C01825=1176.377,-89.170,-41.467,179.123,5.741,149.280
C01826=1176.382,-89.420,-41.456,179.120,5.741,149.280
C01827=1176.387,-89.669,-41.446,179.119,5.741,149.281
C01828=1176.393,-89.919,-41.437,179.116,5.740,149.282
C01829=1176.399,-90.169,-41.427,179.114,5.739,149.282
C01830=1176.403,-90.419,-41.417,179.112,5.740,149.283
C01831=1176.409,-90.668,-41.406,179.110,5.739,149.283
C01832=1176.414,-90.918,-41.396,179.108,5.739,149.284
C01833=1176.419,-91.168,-41.387,179.105,5.739,149.285
C01834=1176.424,-91.418,-41.377,179.103,5.738,149.285
C01835=1176.430,-91.668,-41.367,179.101,5.739,149.286
C01836=1176.435,-91.917,-41.357,179.098,5.738,149.286
C01837=1176.441,-92.167,-41.347,179.096,5.738,149.287
C01838=1176.446,-92.417,-41.337,179.094,5.738,149.288
C01839=1176.451,-92.666,-41.327,179.092,5.737,149.288
C01840=1176.456,-92.916,-41.317,179.090,5.737,149.289
C01841=1176.462,-93.166,-41.308,179.087,5.737,149.290
C01842=1176.467,-93.415,-41.298,179.086,5.737,149.290
C01843=1176.472,-93.666,-41.287,179.083,5.736,149.291
C01844=1176.478,-93.915,-41.277,179.081,5.736,149.291
C01845=1176.483,-94.165,-41.268,179.079,5.736,149.292
C01846=1176.488,-94.415,-41.258,179.077,5.735,149.292
C01847=1176.493,-94.664,-41.248,179.074,5.736,149.293
C01848=1176.499,-94.915,-41.239,179.072,5.735,149.294
C01849=1176.504,-95.164,-41.228,179.070,5.734,149.294
C01850=1176.509,-95.413,-41.219,179.068,5.734,149.295
C01851=1176.515,-95.664,-41.209,179.065,5.734,149.296
C01852=1176.520,-95.913,-41.200,179.064,5.734,149.296
C01853=1176.525,-96.162,-41.189,179.061,5.734,149.297
C01854=1176.531,-96.413,-41.180,179.059,5.734,149.297
C01855=1176.536,-96.663,-41.170,179.057,5.733,149.298
C01856=1176.541,-96.912,-41.160,179.055,5.733,149.298
C01857=1176.546,-97.162,-41.151,179.053,5.733,149.299
C01858=1176.552,-97.411,-41.141,179.050,5.732,149.300
C01859=1176.557,-97.661,-41.132,179.048,5.733,149.300
C01860=1176.562,-97.912,-41.121,179.046,5.732,149.301
C01861=1176.568,-98.161,-41.111,179.044,5.732,149.302
C01862=1176.573,-98.411,-41.102,179.042,5.731,149.302
C01863=1176.578,-98.660,-41.092,179.039,5.731,149.303
C01864=1176.584,-98.910,-41.083,179.038,5.731,149.303
C01865=1176.589,-99.160,-41.073,179.035,5.731,149.304
C01866=1176.594,-99.410,-41.064,179.033,5.731,149.304
C01867=1176.600,-99.659,-41.054,179.031,5.730,149.305
C01868=1176.604,-99.909,-41.044,179.029,5.730,149.306
C01869=1176.610,-100.159,-41.034,179.026,5.730,149.306
C01870=1176.615,-100.409,-41.025,179.024,5.729,149.307
C01871=1176.621,-100.659,-41.015,179.022,5.729,149.308
C01872=1176.626,-100.908,-41.005,179.020,5.729,149.308
C01873=1176.632,-101.158,-40.996,179.018,5.729,149.309
C01874=1176.636,-101.407,-40.986,179.016,5.728,149.309
C01875=1176.643,-101.680,-40.976,179.013,5.728,149.310
C01876=1176.648,-101.952,-40.965,179.011,5.728,149.311
C01877=1176.654,-102.223,-40.955,179.009,5.728,149.311
C01878=1176.660,-102.495,-40.945,179.006,5.727,149.312
C01879=1176.665,-102.745,-40.935,179.004,5.728,149.313
C01880=1176.670,-102.995,-40.926,179.002,5.727,149.313
C01881=1176.676,-103.244,-40.916,179.000,5.727,149.314
C01882=1176.681,-103.494,-40.907,178.997,5.726,149.314
C01883=1176.686,-103.743,-40.897,178.996,5.726,149.315
C01884=1176.691,-103.994,-40.888,178.993,5.726,149.315
C01885=1176.696,-104.243,-40.878,178.992,5.726,149.316
C01886=1176.702,-104.493,-40.868,178.989,5.726,149.317
C01887=1176.707,-104.743,-40.860,178.987,5.725,149.317
C01888=1176.713,-104.992,-40.849,178.985,5.725,149.318
C01889=1176.718,-105.242,-40.840,178.982,5.725,149.318
C01890=1176.723,-105.491,-40.831,178.980,5.725,149.319
C01891=1176.729,-105.742,-40.821,178.978,5.724,149.319
C01892=1176.734,-105.991,-40.812,178.976,5.725,149.320
C01893=1176.740,-106.241,-40.802,178.974,5.724,149.321
C01894=1176.745,-106.491,-40.793,178.972,5.724,149.321
C01895=1176.749,-106.741,-40.783,178.970,5.723,149.322
C01896=1176.755,-106.991,-40.774,178.967,5.723,149.323
C01897=1176.760,-107.241,-40.765,178.965,5.723,149.323
C01898=1176.765,-107.490,-40.755,178.963,5.723,149.324
C01899=1176.771,-107.740,-40.746,178.961,5.723,149.324
C01900=1176.776,-107.990,-40.737,178.959,5.722,149.325
C01901=1176.781,-108.239,-40.727,178.957,5.722,149.325
C01902=1176.787,-108.489,-40.718,178.955,5.722,149.326
C01903=1176.792,-108.739,-40.709,178.952,5.722,149.327
C01904=1176.797,-108.989,-40.699,178.950,5.721,149.327
C01905=1176.803,-109.239,-40.690,178.948,5.722,149.328
C01906=1176.808,-109.489,-40.681,178.946,5.721,149.328
C01907=1176.813,-109.738,-40.672,178.944,5.721,149.329
C01908=1176.819,-109.988,-40.662,178.942,5.721,149.330
C01909=1176.824,-110.238,-40.653,178.940,5.721,149.330
C01910=1176.829,-110.488,-40.644,178.937,5.720,149.331
C01911=1176.835,-110.737,-40.634,178.935,5.719,149.331
C01912=1176.840,-110.987,-40.625,178.933,5.720,149.332
C01913=1176.845,-111.237,-40.616,178.931,5.719,149.332
C01914=1176.851,-111.487,-40.607,178.929,5.719,149.333
C01915=1176.856,-111.737,-40.598,178.927,5.719,149.334
C01916=1176.862,-111.985,-40.588,178.925,5.719,149.334
C01917=1176.867,-112.235,-40.579,178.922,5.718,149.335
C01918=1176.873,-112.485,-40.570,178.920,5.719,149.336
C01919=1176.878,-112.735,-40.561,178.918,5.718,149.336
C01920=1176.883,-112.985,-40.551,178.917,5.718,149.337
C01921=1176.889,-113.235,-40.542,178.914,5.718,149.337
C01922=1176.894,-113.485,-40.533,178.912,5.718,149.338
C01923=1176.899,-113.734,-40.524,178.910,5.717,149.338
C01924=1176.904,-113.984,-40.515,178.908,5.717,149.339
C01925=1176.910,-114.234,-40.506,178.905,5.717,149.340
C01926=1176.915,-114.484,-40.496,178.904,5.717,149.340
C01927=1176.920,-114.733,-40.487,178.901,5.716,149.341
C01928=1176.925,-114.983,-40.478,178.899,5.717,149.341
C01929=1176.931,-115.234,-40.469,178.897,5.716,149.342
C01930=1176.936,-115.483,-40.460,178.895,5.716,149.343
C01931=1176.941,-115.733,-40.451,178.893,5.715,149.343
C01932=1176.947,-115.982,-40.442,178.891,5.716,149.344
C01933=1176.952,-116.232,-40.433,178.889,5.715,149.344
C01934=1176.958,-116.482,-40.423,178.886,5.714,149.345
C01935=1176.963,-116.732,-40.415,178.884,5.715,149.345
C01936=1176.968,-116.981,-40.406,178.882,5.714,149.346
C01937=1176.973,-117.231,-40.397,178.880,5.714,149.347
C01938=1176.979,-117.481,-40.388,178.878,5.714,149.347
C01939=1176.984,-117.731,-40.379,178.876,5.714,149.348
C01940=1176.990,-117.981,-40.369,178.874,5.713,149.348
C01941=1176.995,-118.231,-40.361,178.872,5.713,149.349
C01942=1177.001,-118.480,-40.352,178.869,5.713,149.350
C01943=1177.006,-118.730,-40.343,178.868,5.713,149.350
C01944=1177.011,-118.979,-40.334,178.865,5.713,149.351
C01945=1177.016,-119.229,-40.325,178.863,5.713,149.351
C01946=1177.022,-119.479,-40.315,178.861,5.712,149.352
C01947=1177.027,-119.729,-40.306,178.859,5.712,149.352
C01948=1177.032,-119.979,-40.297,178.857,5.711,149.353
C01949=1177.037,-120.229,-40.288,178.855,5.712,149.354
C01950=1177.043,-120.478,-40.280,178.853,5.711,149.354
C01951=1177.048,-120.728,-40.271,178.851,5.711,149.355
C01952=1177.053,-120.978,-40.262,178.848,5.711,149.355
C01953=1177.058,-121.228,-40.253,178.847,5.711,149.356
C01954=1177.064,-121.477,-40.244,178.844,5.710,149.357
C01955=1177.070,-121.728,-40.235,178.843,5.710,149.357
C01956=1177.075,-121.977,-40.226,178.840,5.710,149.357
C01957=1177.080,-122.227,-40.217,178.838,5.710,149.358
C01958=1177.086,-122.476,-40.209,178.836,5.709,149.359
C01959=1177.091,-122.726,-40.200,178.834,5.710,149.359
C01960=1177.096,-122.977,-40.191,178.832,5.709,149.360
C01961=1177.101,-123.227,-40.183,178.830,5.709,149.360
C01962=1177.107,-123.476,-40.174,178.828,5.709,149.361
C01963=1177.112,-123.726,-40.165,178.826,5.709,149.362
C01964=1177.118,-123.975,-40.156,178.824,5.709,149.362
C01965=1177.123,-124.225,-40.147,178.822,5.708,149.363
C01966=1177.128,-124.475,-40.138,178.820,5.708,149.363
C01967=1177.133,-124.725,-40.130,178.817,5.708,149.364
C01968=1177.139,-124.974,-40.121,178.816,5.708,149.364
C01969=1177.144,-125.224,-40.112,178.814,5.707,149.365
C01970=1177.150,-125.474,-40.103,178.812,5.708,149.366
C01971=1177.155,-125.724,-40.094,178.809,5.707,149.366
C01972=1177.161,-125.974,-40.086,178.807,5.707,149.367
C01973=1177.166,-126.224,-40.077,178.805,5.706,149.367
C01974=1177.171,-126.473,-40.068,178.803,5.706,149.368
C01975=1177.177,-126.723,-40.059,178.801,5.706,149.369
C01976=1177.182,-126.973,-40.050,178.799,5.706,149.369
C01977=1177.188,-127.222,-40.042,178.797,5.705,149.370
C01978=1177.193,-127.473,-40.034,178.795,5.706,149.370
C01979=1176.771,-127.484,-40.074,178.791,5.709,149.372
C01980=1176.766,-127.234,-40.083,178.793,5.709,149.371
C01981=1176.761,-126.984,-40.091,178.795,5.709,149.371
C01982=1176.756,-126.734,-40.100,178.797,5.709,149.370
C01983=1176.750,-126.485,-40.108,178.800,5.710,149.370
C01984=1176.745,-126.235,-40.117,178.801,5.710,149.369
C01985=1176.739,-125.985,-40.126,178.803,5.710,149.369
C01986=1176.734,-125.735,-40.135,178.805,5.710,149.368
C01987=1176.729,-125.485,-40.144,178.808,5.711,149.368
C01988=1176.723,-125.236,-40.152,178.810,5.710,149.367
C01989=1176.718,-124.986,-40.160,178.812,5.711,149.366
C01990=1176.713,-124.736,-40.169,178.814,5.711,149.366
C01991=1176.707,-124.486,-40.179,178.816,5.711,149.365
C01992=1176.702,-124.236,-40.188,178.818,5.711,149.365
C01993=1176.696,-123.987,-40.196,178.820,5.712,149.364
C01994=1176.691,-123.737,-40.205,178.822,5.712,149.363
C01995=1176.685,-123.487,-40.214,178.824,5.713,149.363
C01996=1176.680,-123.237,-40.223,178.826,5.712,149.362
C01997=1176.675,-122.987,-40.232,178.829,5.713,149.362
C01998=1176.670,-122.737,-40.241,178.830,5.713,149.361
C01999=1176.664,-122.488,-40.249,178.833,5.713,149.361
C02000=1176.659,-122.238,-40.257,178.834,5.713,149.360
C02001=1176.654,-121.988,-40.266,178.837,5.714,149.360
C02002=1176.648,-121.738,-40.275,178.839,5.714,149.359
C02003=1176.643,-121.488,-40.284,178.841,5.714,149.358
C02004=1176.638,-121.238,-40.293,178.843,5.714,149.358
C02005=1176.632,-120.989,-40.302,178.845,5.715,149.357
C02006=1176.626,-120.739,-40.311,178.847,5.715,149.357
C02007=1176.621,-120.489,-40.320,178.849,5.715,149.356
C02008=1176.616,-120.239,-40.329,178.851,5.715,149.355
C02009=1176.611,-119.990,-40.338,178.854,5.715,149.355
C02010=1176.606,-119.740,-40.347,178.855,5.715,149.354
C02011=1176.601,-119.490,-40.356,178.858,5.716,149.354
C02012=1176.595,-119.241,-40.364,178.860,5.716,149.353
C02013=1176.589,-118.991,-40.374,178.862,5.717,149.353
C02014=1176.584,-118.741,-40.383,178.864,5.716,149.352
C02015=1176.579,-118.491,-40.392,178.866,5.717,149.351
C02016=1176.574,-118.242,-40.401,178.868,5.717,149.351
C02017=1176.569,-117.992,-40.410,178.870,5.717,149.350
C02018=1176.563,-117.742,-40.419,178.872,5.717,149.350
C02019=1176.558,-117.492,-40.428,178.875,5.718,149.349
C02020=1176.552,-117.242,-40.437,178.876,5.718,149.348
C02021=1176.547,-116.993,-40.446,178.879,5.718,149.348
C02022=1176.541,-116.743,-40.455,178.880,5.718,149.347
C02023=1176.536,-116.493,-40.464,178.883,5.719,149.347
C02024=1176.531,-116.243,-40.472,178.885,5.718,149.346
C02025=1176.525,-115.993,-40.482,178.887,5.719,149.346
C02026=1176.520,-115.744,-40.492,178.889,5.719,149.345
C02027=1176.515,-115.494,-40.500,178.891,5.719,149.344
C02028=1176.510,-115.244,-40.509,178.893,5.719,149.344
C02029=1176.505,-114.994,-40.518,178.896,5.720,149.343
C02030=1176.499,-114.744,-40.528,178.897,5.720,149.343
C02031=1176.494,-114.494,-40.537,178.900,5.720,149.342
C02032=1176.488,-114.245,-40.545,178.901,5.720,149.342
C02033=1176.483,-113.996,-40.555,178.904,5.720,149.341
C02034=1176.477,-113.746,-40.564,178.906,5.720,149.340
C02035=1176.472,-113.496,-40.573,178.908,5.721,149.340
C02036=1176.467,-113.246,-40.582,178.910,5.721,149.339
C02037=1176.462,-112.996,-40.591,178.912,5.722,149.339
C02038=1176.456,-112.747,-40.601,178.914,5.721,149.338
C02039=1176.451,-112.497,-40.610,178.916,5.722,149.337
C02040=1176.446,-112.247,-40.619,178.919,5.722,149.337
C02041=1176.440,-111.997,-40.628,178.921,5.722,149.336
C02042=1176.435,-111.747,-40.637,178.923,5.723,149.336
C02043=1176.430,-111.498,-40.647,178.925,5.723,149.335
C02044=1176.425,-111.248,-40.656,178.927,5.723,149.335
C02045=1176.419,-110.998,-40.665,178.929,5.723,149.334
C02046=1176.414,-110.748,-40.674,178.931,5.724,149.333
C02047=1176.409,-110.499,-40.684,178.934,5.723,149.333
C02048=1176.403,-110.248,-40.693,178.936,5.724,149.332
C02049=1176.398,-109.999,-40.702,178.938,5.724,149.331
C02050=1176.392,-109.749,-40.711,178.940,5.725,149.331
C02051=1176.387,-109.499,-40.721,178.942,5.724,149.330
C02052=1176.382,-109.249,-40.730,178.944,5.725,149.330
C02053=1176.377,-108.999,-40.739,178.946,5.725,149.329
C02054=1176.371,-108.750,-40.749,178.949,5.725,149.329
C02055=1176.366,-108.500,-40.758,178.951,5.726,149.328
C02056=1176.361,-108.250,-40.767,178.953,5.726,149.327
C02057=1176.355,-108.001,-40.777,178.955,5.726,149.327
C02058=1176.350,-107.751,-40.786,178.957,5.726,149.326
C02059=1176.345,-107.501,-40.795,178.959,5.727,149.326
C02060=1176.339,-107.251,-40.805,178.961,5.726,149.325
C02061=1176.334,-107.002,-40.814,178.964,5.727,149.324
C02062=1176.329,-106.752,-40.823,178.965,5.727,149.324
C02063=1176.323,-106.502,-40.833,178.968,5.727,149.323
C02064=1176.318,-106.252,-40.842,178.969,5.727,149.323
C02065=1176.313,-106.002,-40.851,178.972,5.728,149.322
C02066=1176.307,-105.753,-40.861,178.974,5.728,149.322
C02067=1176.302,-105.503,-40.870,178.976,5.728,149.321
C02068=1176.296,-105.254,-40.880,178.979,5.729,149.320
C02069=1176.291,-105.004,-40.889,178.981,5.729,149.320
C02070=1176.286,-104.754,-40.898,178.983,5.729,149.319
C02071=1176.281,-104.504,-40.909,178.985,5.729,149.318
C02072=1176.275,-104.254,-40.917,178.987,5.730,149.318
C02073=1176.270,-104.005,-40.928,178.989,5.729,149.317
C02074=1176.265,-103.754,-40.937,178.991,5.730,149.317
C02075=1176.260,-103.505,-40.947,178.993,5.730,149.316
C02076=1176.254,-103.255,-40.956,178.996,5.730,149.316
C02077=1176.249,-103.005,-40.965,178.998,5.731,149.315
C02078=1176.244,-102.756,-40.975,179.000,5.731,149.314
C02079=1176.239,-102.506,-40.984,179.002,5.732,149.314
C02080=1176.232,-102.233,-40.995,179.004,5.731,149.313
C02081=1176.226,-101.963,-41.005,179.007,5.732,149.312
C02082=1176.221,-101.691,-41.016,179.010,5.732,149.312
C02083=1176.216,-101.419,-41.026,179.011,5.732,149.311
C02084=1176.210,-101.169,-41.035,179.014,5.732,149.311
C02085=1176.205,-100.920,-41.045,179.016,5.733,149.310
C02086=1176.199,-100.669,-41.054,179.018,5.733,149.309
C02087=1176.194,-100.420,-41.064,179.020,5.733,149.309
C02088=1176.189,-100.170,-41.075,179.022,5.733,149.308
C02089=1176.184,-99.920,-41.084,179.025,5.734,149.308
C02090=1176.178,-99.671,-41.094,179.027,5.733,149.307
C02091=1176.173,-99.421,-41.103,179.029,5.734,149.306
C02092=1176.167,-99.171,-41.113,179.032,5.735,149.306
C02093=1176.162,-98.921,-41.122,179.033,5.735,149.305
C02094=1176.157,-98.672,-41.132,179.036,5.735,149.305
C02095=1176.152,-98.422,-41.141,179.037,5.735,149.304
C02096=1176.147,-98.172,-41.151,179.040,5.735,149.303
C02097=1176.142,-97.922,-41.161,179.042,5.735,149.303
C02098=1176.136,-97.672,-41.171,179.044,5.736,149.302
C02099=1176.130,-97.423,-41.181,179.047,5.737,149.302
C02100=1176.125,-97.173,-41.190,179.049,5.736,149.301
C02101=1176.119,-96.923,-41.200,179.051,5.737,149.300
C02102=1176.115,-96.674,-41.209,179.053,5.736,149.300
C02103=1176.109,-96.423,-41.219,179.055,5.737,149.299
C02104=1176.104,-96.174,-41.229,179.057,5.737,149.299
C02105=1176.099,-95.924,-41.239,179.059,5.738,149.298
C02106=1176.093,-95.674,-41.249,179.062,5.738,149.297
C02107=1176.088,-95.425,-41.258,179.064,5.738,149.297
C02108=1176.082,-95.176,-41.268,179.066,5.738,149.296
C02109=1176.078,-94.925,-41.278,179.068,5.738,149.296
C02110=1176.072,-94.675,-41.288,179.071,5.739,149.295
C02111=1176.067,-94.426,-41.298,179.073,5.740,149.295
C02112=1176.061,-94.176,-41.307,179.075,5.739,149.294
C02113=1176.056,-93.927,-41.317,179.077,5.740,149.293
C02114=1176.051,-93.676,-41.328,179.079,5.740,149.293
C02115=1176.046,-93.426,-41.337,179.081,5.740,149.292
C02116=1176.040,-93.177,-41.347,179.083,5.740,149.291
C02117=1176.035,-92.928,-41.357,179.086,5.741,149.291
C02118=1176.030,-92.678,-41.367,179.088,5.741,149.290
C02119=1176.024,-92.427,-41.377,179.090,5.741,149.290
C02120=1176.020,-92.178,-41.386,179.093,5.741,149.289
C02121=1176.014,-91.928,-41.396,179.094,5.741,149.289
C02122=1176.008,-91.679,-41.407,179.097,5.742,149.288
C02123=1176.004,-91.428,-41.416,179.099,5.743,149.287
C02124=1175.998,-91.179,-41.426,179.101,5.742,149.287
C02125=1175.993,-90.929,-41.436,179.103,5.743,149.286
C02126=1175.988,-90.680,-41.446,179.105,5.743,149.285
C02127=1175.982,-90.429,-41.456,179.108,5.743,149.285
C02128=1175.977,-90.180,-41.466,179.110,5.744,149.284
C02129=1175.972,-89.930,-41.476,179.112,5.743,149.284
C02130=1175.966,-89.681,-41.486,179.114,5.744,149.283
C02131=1175.961,-89.431,-41.496,179.117,5.744,149.282
C02132=1175.955,-89.180,-41.506,179.119,5.745,149.282
C02133=1175.951,-88.931,-41.515,179.121,5.745,149.281
C02134=1175.945,-88.682,-41.526,179.123,5.745,149.281
C02135=1175.940,-88.431,-41.536,179.126,5.745,149.280
C02136=1175.935,-88.182,-41.546,179.127,5.745,149.279
C02137=1175.930,-87.933,-41.556,179.130,5.746,149.279
C02138=1175.924,-87.683,-41.566,179.132,5.747,149.278
C02139=1175.919,-87.432,-41.576,179.134,5.746,149.278
C02140=1175.914,-87.183,-41.586,179.136,5.747,149.277
C02141=1175.908,-86.933,-41.596,179.139,5.747,149.276
C02142=1175.903,-86.683,-41.607,179.141,5.747,149.276
C02143=1175.898,-86.434,-41.617,179.143,5.748,149.275
C02144=1175.893,-86.184,-41.626,179.145,5.747,149.274
C02145=1175.888,-85.934,-41.637,179.148,5.748,149.274
C02146=1175.882,-85.685,-41.647,179.150,5.748,149.273
C02147=1175.876,-85.435,-41.657,179.152,5.748,149.273
C02148=1175.871,-85.186,-41.668,179.155,5.749,149.272
C02149=1175.867,-84.936,-41.678,179.157,5.750,149.272
C02150=1175.861,-84.686,-41.688,179.159,5.749,149.271
C02151=1175.855,-84.437,-41.698,179.161,5.750,149.270
C02152=1175.850,-84.186,-41.708,179.163,5.750,149.270
C02153=1175.845,-83.936,-41.718,179.165,5.750,149.269
C02154=1175.840,-83.687,-41.728,179.168,5.751,149.269
C02155=1175.835,-83.437,-41.738,179.170,5.750,149.268
C02156=1175.829,-83.187,-41.748,179.172,5.751,149.267
C02157=1175.823,-82.938,-41.759,179.175,5.752,149.267
C02158=1175.818,-82.687,-41.769,179.177,5.752,149.266
C02159=1175.813,-82.438,-41.779,179.179,5.752,149.265
C02160=1175.809,-82.188,-41.789,179.181,5.752,149.265
C02161=1175.803,-81.938,-41.800,179.183,5.752,149.264
C02162=1175.798,-81.689,-41.811,179.186,5.753,149.264
C02163=1175.793,-81.439,-41.821,179.188,5.753,149.263
C02164=1175.787,-81.190,-41.831,179.190,5.754,149.263
C02165=1175.782,-80.940,-41.842,179.193,5.754,149.262
C02166=1175.777,-80.690,-41.852,179.195,5.754,149.261
C02167=1175.771,-80.440,-41.862,179.197,5.754,149.261
C02168=1175.766,-80.191,-41.872,179.200,5.755,149.260
C02169=1175.761,-79.941,-41.883,179.201,5.755,149.259
C02170=1175.755,-79.691,-41.893,179.204,5.755,149.259
C02171=1175.750,-79.441,-41.903,179.205,5.755,149.258
C02172=1175.745,-79.191,-41.914,179.208,5.756,149.258
C02173=1175.739,-78.942,-41.924,179.211,5.756,149.257
C02174=1175.734,-78.692,-41.934,179.212,5.756,149.256
C02175=1175.729,-78.443,-41.945,179.215,5.756,149.256
C02176=1175.724,-78.193,-41.956,179.217,5.757,149.255
C02177=1175.718,-77.943,-41.966,179.219,5.757,149.254
C02178=1175.713,-77.693,-41.976,179.221,5.758,149.254
C02179=1175.708,-77.443,-41.987,179.224,5.758,149.253
C02180=1175.702,-77.194,-41.997,179.226,5.758,149.253
C02181=1175.697,-76.943,-42.008,179.228,5.758,149.252
C02182=1175.692,-76.694,-42.018,179.231,5.759,149.251
C02183=1175.687,-76.444,-42.029,179.233,5.759,149.251
C02184=1175.681,-76.174,-42.040,179.235,5.759,149.250
C02185=1175.675,-75.902,-42.051,179.238,5.760,149.249
C02186=1175.670,-75.632,-42.062,179.241,5.760,149.249
C02187=1175.664,-75.360,-42.074,179.242,5.760,149.248
C02188=1175.659,-75.110,-42.085,179.245,5.760,149.248
C02189=1175.654,-74.861,-42.095,179.247,5.761,149.247
C02190=1175.649,-74.611,-42.106,179.249,5.761,149.246
C02191=1175.643,-74.361,-42.116,179.252,5.761,149.246
C02192=1175.637,-74.112,-42.126,179.254,5.762,149.245
C02193=1175.632,-73.862,-42.137,179.256,5.762,149.245
C02194=1175.627,-73.613,-42.148,179.258,5.762,149.244
C02195=1175.622,-73.363,-42.159,179.261,5.763,149.243
C02196=1175.616,-73.113,-42.169,179.263,5.762,149.243
C02197=1175.612,-72.863,-42.180,179.265,5.763,149.242
C02198=1175.606,-72.614,-42.190,179.268,5.764,149.241
C02199=1175.601,-72.364,-42.201,179.270,5.764,149.241
C02200=1175.596,-72.114,-42.211,179.272,5.764,149.240
C02201=1175.591,-71.864,-42.222,179.274,5.765,149.240
C02202=1175.585,-71.615,-42.233,179.276,5.764,149.239
C02203=1175.580,-71.364,-42.244,179.279,5.765,149.238
C02204=1175.574,-71.115,-42.255,179.281,5.766,149.238
C02205=1175.569,-70.865,-42.265,179.283,5.765,149.237
C02206=1175.564,-70.616,-42.275,179.286,5.766,149.237
C02207=1175.559,-70.366,-42.287,179.288,5.766,149.236
C02208=1175.553,-70.116,-42.297,179.291,5.767,149.235
C02209=1175.548,-69.866,-42.307,179.293,5.767,149.235
C02210=1175.543,-69.617,-42.318,179.295,5.767,149.234
C02211=1175.538,-69.367,-42.329,179.297,5.768,149.234
C02212=1175.533,-69.118,-42.340,179.299,5.768,149.233
C02213=1175.527,-68.868,-42.351,179.302,5.768,149.232
C02214=1175.521,-68.618,-42.361,179.304,5.769,149.232
C02215=1175.517,-68.368,-42.373,179.306,5.768,149.231
C02216=1175.511,-68.119,-42.383,179.309,5.769,149.231
C02217=1175.506,-67.869,-42.394,179.311,5.770,149.230
C02218=1175.501,-67.619,-42.405,179.313,5.770,149.229
C02219=1175.496,-67.369,-42.415,179.316,5.770,149.229
C02220=1175.490,-67.119,-42.427,179.318,5.770,149.228
C02221=1175.485,-66.870,-42.437,179.320,5.770,149.227
C02222=1175.480,-66.620,-42.448,179.322,5.771,149.227
C02223=1175.475,-66.371,-42.458,179.325,5.772,149.226
C02224=1175.470,-66.121,-42.470,179.327,5.772,149.226
C02225=1175.465,-65.871,-42.480,179.329,5.772,149.225
C02226=1175.459,-65.622,-42.492,179.332,5.773,149.224
C02227=1175.454,-65.371,-42.502,179.334,5.773,149.224
C02228=1175.449,-65.122,-42.513,179.336,5.773,149.223
C02229=1175.444,-64.872,-42.524,179.339,5.773,149.222
C02230=1175.438,-64.623,-42.535,179.341,5.774,149.222
C02231=1175.433,-64.373,-42.546,179.343,5.774,149.221
C02232=1175.428,-64.123,-42.557,179.345,5.774,149.221
C02233=1175.422,-63.874,-42.568,179.348,5.775,149.220
C02234=1175.418,-63.624,-42.579,179.350,5.775,149.219
C02235=1175.411,-63.374,-42.590,179.352,5.775,149.219
C02236=1175.406,-63.124,-42.601,179.355,5.776,149.218
C02237=1175.402,-62.875,-42.612,179.357,5.776,149.217
C02238=1175.396,-62.625,-42.622,179.359,5.776,149.217
C02239=1175.391,-62.375,-42.634,179.361,5.777,149.216
C02240=1175.386,-62.125,-42.645,179.364,5.777,149.216
C02241=1175.380,-61.876,-42.656,179.366,5.778,149.215
C02242=1175.376,-61.627,-42.667,179.368,5.777,149.214
C02243=1175.370,-61.376,-42.678,179.371,5.778,149.214
C02244=1175.365,-61.127,-42.689,179.373,5.779,149.213
C02245=1175.360,-60.877,-42.700,179.375,5.778,149.213
C02246=1175.354,-60.628,-42.711,179.378,5.779,149.212
C02247=1175.349,-60.378,-42.723,179.380,5.780,149.211
C02248=1175.344,-60.128,-42.733,179.382,5.780,149.211
C02249=1175.339,-59.879,-42.744,179.384,5.780,149.210
C02250=1175.333,-59.629,-42.756,179.387,5.780,149.209
C02251=1175.328,-59.379,-42.767,179.389,5.781,149.209
C02252=1175.323,-59.130,-42.777,179.392,5.782,149.208
C02253=1175.318,-58.880,-42.789,179.394,5.781,149.208
C02254=1175.313,-58.630,-42.800,179.396,5.782,149.207
C02255=1175.308,-58.380,-42.811,179.399,5.782,149.206
C02256=1175.302,-58.131,-42.823,179.400,5.782,149.206
C02257=1175.297,-57.880,-42.833,179.403,5.783,149.205
C02258=1175.292,-57.631,-42.845,179.406,5.783,149.205
C02259=1175.286,-57.382,-42.856,179.408,5.784,149.204
C02260=1175.281,-57.132,-42.867,179.410,5.784,149.203
C02261=1175.276,-56.882,-42.878,179.412,5.784,149.203
C02262=1175.270,-56.632,-42.889,179.415,5.785,149.202
C02263=1175.266,-56.383,-42.901,179.418,5.785,149.201
C02264=1175.261,-56.133,-42.912,179.419,5.785,149.201
C02265=1175.255,-55.883,-42.923,179.422,5.786,149.200
C02266=1175.250,-55.634,-42.934,179.425,5.786,149.200
C02267=1175.245,-55.384,-42.946,179.427,5.787,149.199
C02268=1175.240,-55.134,-42.957,179.429,5.787,149.198
C02269=1175.235,-54.885,-42.969,179.431,5.787,149.198
C02270=1175.229,-54.635,-42.979,179.434,5.788,149.197
C02271=1175.224,-54.385,-42.991,179.436,5.788,149.196
C02272=1175.219,-54.135,-43.003,179.438,5.788,149.196
C02273=1175.214,-53.886,-43.014,179.441,5.789,149.195
C02274=1175.208,-53.636,-43.025,179.443,5.789,149.195
C02275=1175.203,-53.387,-43.037,179.445,5.790,149.194
C02276=1175.198,-53.136,-43.047,179.448,5.790,149.193
C02277=1175.193,-52.886,-43.059,179.450,5.790,149.193
C02278=1175.188,-52.638,-43.070,179.452,5.791,149.192
C02279=1175.182,-52.388,-43.082,179.455,5.791,149.192
C02280=1175.178,-52.138,-43.093,179.457,5.791,149.191
C02281=1175.172,-51.888,-43.105,179.459,5.792,149.190
C02282=1175.167,-51.639,-43.116,179.461,5.792,149.190
C02283=1175.161,-51.389,-43.128,179.464,5.793,149.189
C02284=1175.157,-51.140,-43.139,179.466,5.792,149.188
C02285=1175.151,-50.889,-43.150,179.468,5.793,149.188
C02286=1175.146,-50.639,-43.162,179.471,5.794,149.187
C02287=1175.140,-50.390,-43.173,179.474,5.794,149.187
C02288=1175.135,-50.120,-43.186,179.476,5.795,149.186
C02289=1175.129,-49.849,-43.198,179.479,5.795,149.185
C02290=1175.123,-49.579,-43.211,179.481,5.795,149.185
C02291=1175.118,-49.308,-43.223,179.483,5.795,149.184
C02292=1175.113,-49.059,-43.235,179.486,5.796,149.183
C02293=1175.108,-48.809,-43.246,179.488,5.797,149.183
C02294=1175.102,-48.560,-43.257,179.491,5.797,149.182
C02295=1175.097,-48.310,-43.269,179.492,5.797,149.182
C02296=1175.092,-48.060,-43.281,179.495,5.797,149.181
C02297=1175.087,-47.810,-43.292,179.498,5.798,149.180
C02298=1175.082,-47.561,-43.304,179.500,5.799,149.180
C02299=1175.077,-47.311,-43.316,179.503,5.799,149.179
C02300=1175.071,-47.061,-43.327,179.505,5.799,149.178
C02301=1175.066,-46.812,-43.338,179.507,5.800,149.178
C02302=1175.061,-46.562,-43.350,179.510,5.800,149.177
C02303=1175.056,-46.313,-43.362,179.512,5.800,149.176
C02304=1175.051,-46.063,-43.374,179.514,5.800,149.176
C02305=1175.045,-45.813,-43.386,179.516,5.801,149.175
C02306=1175.040,-45.564,-43.397,179.519,5.802,149.175
C02307=1175.035,-45.314,-43.409,179.521,5.802,149.174
C02308=1175.030,-45.064,-43.420,179.524,5.802,149.173
C02309=1175.024,-44.815,-43.432,179.526,5.803,149.173
C02310=1175.019,-44.565,-43.444,179.528,5.803,149.172
C02311=1175.014,-44.315,-43.455,179.531,5.803,149.172
C02312=1175.009,-44.065,-43.467,179.533,5.804,149.171
C02313=1175.004,-43.816,-43.480,179.536,5.805,149.170
C02314=1174.999,-43.566,-43.491,179.538,5.804,149.170
C02315=1174.993,-43.317,-43.503,179.540,5.805,149.169
C02316=1174.988,-43.067,-43.514,179.543,5.805,149.169
C02317=1174.983,-42.817,-43.526,179.545,5.806,149.168
C02318=1174.977,-42.567,-43.538,179.548,5.807,149.167
C02319=1174.972,-42.317,-43.549,179.550,5.806,149.167
C02320=1174.968,-42.068,-43.561,179.552,5.807,149.166
C02321=1174.962,-41.818,-43.573,179.554,5.808,149.165
C02322=1174.957,-41.569,-43.585,179.557,5.808,149.165
C02323=1174.952,-41.319,-43.597,179.559,5.809,149.164
C02324=1174.947,-41.069,-43.608,179.561,5.808,149.164
C02325=1174.942,-40.820,-43.621,179.564,5.809,149.163
C02326=1174.936,-40.570,-43.633,179.566,5.810,149.162
C02327=1174.931,-40.320,-43.644,179.569,5.810,149.162
C02328=1174.925,-40.071,-43.656,179.571,5.811,149.161
C02329=1174.920,-39.822,-43.668,179.574,5.811,149.161
C02330=1174.916,-39.572,-43.680,179.576,5.811,149.160
C02331=1174.910,-39.322,-43.692,179.578,5.812,149.159
C02332=1174.905,-39.072,-43.703,179.581,5.812,149.159
C02333=1174.900,-38.823,-43.716,179.583,5.813,149.158
C02334=1174.894,-38.573,-43.728,179.585,5.813,149.157
C02335=1174.889,-38.323,-43.739,179.588,5.813,149.157
C02336=1174.884,-38.074,-43.752,179.590,5.814,149.156
C02337=1174.879,-37.824,-43.764,179.592,5.814,149.156
C02338=1174.874,-37.574,-43.776,179.595,5.815,149.155
C02339=1174.869,-37.325,-43.788,179.598,5.815,149.154
C02340=1174.864,-37.075,-43.799,179.600,5.816,149.154
C02341=1174.858,-36.825,-43.811,179.602,5.816,149.153
C02342=1174.853,-36.576,-43.824,179.604,5.817,149.153
C02343=1174.848,-36.326,-43.836,179.607,5.817,149.152
C02344=1174.842,-36.076,-43.848,179.609,5.817,149.151
C02345=1174.838,-35.827,-43.860,179.612,5.818,149.151
C02346=1174.832,-35.577,-43.872,179.614,5.819,149.150
C02347=1174.827,-35.327,-43.883,179.616,5.818,149.149
C02348=1174.822,-35.078,-43.896,179.619,5.819,149.149
C02349=1174.816,-34.828,-43.908,179.621,5.820,149.148
C02350=1174.811,-34.578,-43.921,179.624,5.820,149.147
C02351=1174.807,-34.329,-43.932,179.626,5.821,149.147
C02352=1174.801,-34.079,-43.944,179.629,5.821,149.146
C02353=1174.796,-33.830,-43.956,179.631,5.821,149.146
C02354=1174.791,-33.580,-43.968,179.633,5.822,149.145
C02355=1174.786,-33.330,-43.981,179.636,5.822,149.144
C02356=1174.780,-33.080,-43.993,179.638,5.823,149.144
C02357=1174.775,-32.831,-44.005,179.641,5.823,149.143
C02358=1174.770,-32.581,-44.017,179.643,5.824,149.143
C02359=1174.764,-32.332,-44.030,179.645,5.825,149.142
C02360=1174.760,-32.082,-44.041,179.647,5.824,149.141
C02361=1174.755,-31.832,-44.054,179.650,5.825,149.141
C02362=1174.750,-31.582,-44.066,179.652,5.825,149.140
C02363=1174.745,-31.333,-44.079,179.655,5.826,149.139
C02364=1174.739,-31.083,-44.090,179.658,5.826,149.139
C02365=1174.734,-30.834,-44.103,179.660,5.827,149.138
C02366=1174.729,-30.584,-44.115,179.662,5.828,149.138
C02367=1174.724,-30.334,-44.127,179.664,5.827,149.137
C02368=1174.718,-30.084,-44.139,179.667,5.828,149.136
C02369=1174.713,-29.835,-44.152,179.669,5.829,149.136
C02370=1174.708,-29.585,-44.164,179.672,5.829,149.135
C02371=1174.702,-29.336,-44.176,179.674,5.830,149.135
C02372=1174.698,-29.086,-44.189,179.677,5.830,149.134
C02373=1174.693,-28.836,-44.201,179.680,5.831,149.133
C02374=1174.687,-28.587,-44.214,179.681,5.831,149.133
C02375=1174.682,-28.337,-44.226,179.684,5.831,149.132
C02376=1174.677,-28.087,-44.238,179.686,5.832,149.132
C02377=1174.672,-27.838,-44.251,179.689,5.832,149.131
C02378=1174.666,-27.588,-44.263,179.691,5.833,149.130
C02379=1174.661,-27.339,-44.275,179.693,5.834,149.130
C02380=1174.657,-27.089,-44.288,179.696,5.834,149.129
C02381=1174.651,-26.839,-44.300,179.699,5.835,149.128
C02382=1174.646,-26.590,-44.313,179.700,5.835,149.128
C02383=1174.641,-26.340,-44.326,179.703,5.835,149.127
C02384=1174.636,-26.090,-44.337,179.706,5.835,149.126
C02385=1174.630,-25.841,-44.350,179.708,5.836,149.126
C02386=1174.625,-25.592,-44.363,179.711,5.837,149.125
C02387=1174.620,-25.341,-44.375,179.713,5.837,149.125
C02388=1174.615,-25.092,-44.387,179.715,5.838,149.124
C02389=1174.610,-24.842,-44.400,179.718,5.838,149.123
C02390=1174.605,-24.592,-44.412,179.721,5.839,149.123
C02391=1174.600,-24.343,-44.425,179.722,5.839,149.122
C02392=1174.595,-24.073,-44.438,179.725,5.839,149.122
C02393=1174.589,-23.803,-44.453,179.728,5.841,149.121
C02394=1174.583,-23.534,-44.465,179.731,5.841,149.120
C02395=1174.577,-23.264,-44.479,179.734,5.841,149.119
C02396=1174.572,-23.014,-44.492,179.735,5.841,149.119
C02397=1174.567,-22.765,-44.505,179.738,5.842,149.118
C02398=1174.562,-22.514,-44.517,179.740,5.842,149.118
C02399=1174.557,-22.265,-44.529,179.743,5.843,149.117
C02400=1174.552,-22.016,-44.542,179.745,5.844,149.116
C02401=1174.547,-21.766,-44.555,179.748,5.844,149.116
C02402=1174.541,-21.517,-44.568,179.750,5.845,149.115
C02403=1174.536,-21.266,-44.580,179.753,5.845,149.115
C02404=1174.531,-21.017,-44.593,179.755,5.846,149.114
C02405=1174.526,-20.768,-44.605,179.758,5.847,149.113
C02406=1174.521,-20.518,-44.618,179.760,5.847,149.113
C02407=1174.516,-20.268,-44.631,179.762,5.847,149.112
C02408=1174.510,-20.019,-44.644,179.764,5.848,149.112
C02409=1174.505,-19.769,-44.657,179.767,5.848,149.111
C02410=1174.500,-19.519,-44.669,179.769,5.849,149.110
C02411=1174.495,-19.270,-44.681,179.772,5.849,149.110
C02412=1174.490,-19.020,-44.694,179.775,5.850,149.109
C02413=1174.485,-18.771,-44.707,179.777,5.851,149.109
C02414=1174.479,-18.521,-44.720,179.779,5.851,149.108
C02415=1174.475,-18.271,-44.733,179.782,5.851,149.107
C02416=1174.470,-18.022,-44.745,179.784,5.852,149.107
C02417=1174.464,-17.772,-44.758,179.787,5.853,149.106
C02418=1174.459,-17.523,-44.771,179.790,5.853,149.105
C02419=1174.454,-17.273,-44.784,179.791,5.853,149.105
C02420=1174.449,-17.023,-44.797,179.794,5.854,149.104
C02421=1174.444,-16.774,-44.809,179.797,5.854,149.103
C02422=1174.439,-16.524,-44.823,179.799,5.855,149.103
C02423=1174.433,-16.274,-44.836,179.801,5.855,149.102
C02424=1174.428,-16.025,-44.848,179.804,5.856,149.102
C02425=1174.423,-15.776,-44.861,179.806,5.857,149.101
C02426=1174.418,-15.525,-44.874,179.809,5.857,149.100
C02427=1174.413,-15.276,-44.887,179.812,5.858,149.100
C02428=1174.408,-15.027,-44.900,179.814,5.858,149.099
C02429=1174.402,-14.777,-44.913,179.816,5.859,149.099
C02430=1174.397,-14.527,-44.926,179.819,5.859,149.098
C02431=1174.392,-14.278,-44.938,179.821,5.860,149.097
C02432=1174.388,-14.028,-44.951,179.824,5.861,149.097
C02433=1174.382,-13.778,-44.964,179.826,5.861,149.096
C02434=1174.377,-13.529,-44.977,179.829,5.862,149.096
C02435=1174.372,-13.279,-44.990,179.831,5.861,149.095
C02436=1174.366,-13.029,-45.003,179.833,5.862,149.094
C02437=1174.361,-12.780,-45.016,179.836,5.863,149.094
C02438=1174.357,-12.530,-45.029,179.838,5.863,149.093
C02439=1174.351,-12.281,-45.043,179.840,5.864,149.093
C02440=1174.346,-12.032,-45.055,179.843,5.864,149.092
C02441=1174.341,-11.782,-45.068,179.846,5.865,149.091
C02442=1174.336,-11.532,-45.082,179.848,5.866,149.091
C02443=1174.331,-11.282,-45.094,179.851,5.866,149.090
C02444=1174.325,-11.032,-45.108,179.853,5.867,149.089
C02445=1174.320,-10.783,-45.120,179.855,5.867,149.089
C02446=1174.316,-10.534,-45.134,179.858,5.868,149.088
C02447=1174.310,-10.284,-45.147,179.861,5.868,149.087
C02448=1174.305,-10.034,-45.160,179.863,5.869,149.087
C02449=1174.300,-9.784,-45.173,179.866,5.870,149.086
C02450=1174.294,-9.535,-45.186,179.868,5.870,149.086
C02451=1174.290,-9.286,-45.200,179.870,5.871,149.085
C02452=1174.284,-9.036,-45.213,179.873,5.871,149.084
C02453=1174.280,-8.786,-45.226,179.875,5.872,149.084
C02454=1174.274,-8.536,-45.239,179.878,5.873,149.083
C02455=1174.269,-8.287,-45.252,179.881,5.873,149.083
C02456=1174.264,-8.037,-45.266,179.883,5.874,149.082
C02457=1174.259,-7.788,-45.278,179.885,5.874,149.081
C02458=1174.254,-7.538,-45.291,179.888,5.875,149.081
C02459=1174.249,-7.289,-45.305,179.890,5.876,149.080
C02460=1174.244,-7.039,-45.318,179.893,5.876,149.080
C02461=1174.238,-6.789,-45.331,179.895,5.877,149.079
C02462=1174.234,-6.539,-45.344,179.898,5.877,149.078
C02463=1174.228,-6.290,-45.358,179.900,5.877,149.078
C02464=1174.223,-6.041,-45.371,179.902,5.878,149.077
C02465=1174.218,-5.791,-45.385,179.905,5.878,149.077
C02466=1174.213,-5.542,-45.398,179.907,5.879,149.076
C02467=1174.208,-5.292,-45.411,179.910,5.879,149.075
C02468=1174.203,-5.042,-45.424,179.912,5.880,149.075
C02469=1174.198,-4.793,-45.438,179.915,5.881,149.074
C02470=1174.193,-4.543,-45.451,179.917,5.881,149.073
C02471=1174.188,-4.294,-45.465,179.920,5.882,149.073
C02472=1174.182,-4.044,-45.478,179.922,5.882,149.072
C02473=1174.177,-3.794,-45.491,179.924,5.883,149.072
C02474=1174.172,-3.545,-45.505,179.927,5.884,149.071
C02475=1174.167,-3.295,-45.518,179.930,5.884,149.070
C02476=1174.162,-3.046,-45.532,179.932,5.885,149.070
C02477=1174.157,-2.796,-45.545,179.934,5.885,149.069
C02478=1174.151,-2.546,-45.558,179.937,5.886,149.069
C02479=1174.147,-2.297,-45.572,179.939,5.887,149.068
C02480=1174.141,-2.047,-45.585,179.942,5.887,149.067
C02481=1174.136,-1.797,-45.599,179.945,5.888,149.067
C02482=1174.131,-1.548,-45.612,179.947,5.889,149.066
C02483=1174.126,-1.298,-45.626,179.949,5.889,149.066
C02484=1174.121,-1.049,-45.639,179.952,5.889,149.065
C02485=1174.116,-0.799,-45.653,179.954,5.890,149.064
C02486=1174.110,-0.550,-45.666,179.957,5.891,149.064
C02487=1174.106,-0.300,-45.680,179.960,5.891,149.063
C02488=1174.101,-0.050,-45.694,179.962,5.892,149.063
C02489=1174.095,0.199,-45.708,179.965,5.893,149.062
C02490=1174.091,0.449,-45.720,179.967,5.894,149.061
C02491=1174.085,0.698,-45.734,179.970,5.895,149.061
C02492=1174.080,0.948,-45.748,179.972,5.895,149.060
C02493=1174.075,1.197,-45.761,179.975,5.896,149.060
C02494=1174.070,1.447,-45.775,179.977,5.896,149.059
C02495=1174.064,1.696,-45.789,179.980,5.897,149.058
C02496=1174.059,1.965,-45.803,179.983,5.897,149.057
C02497=1174.054,2.235,-45.818,179.985,5.898,149.057
C02498=1174.049,2.504,-45.833,179.987,5.899,149.056
C02499=1174.043,2.773,-45.848,179.990,5.899,149.056
C02500=1174.037,3.023,-45.861,179.993,5.900,149.055
C02501=1174.033,3.273,-45.875,179.995,5.900,149.054
C02502=1174.027,3.522,-45.888,179.998,5.902,149.054
C02503=1174.022,3.772,-45.902,-179.999,5.902,149.053
C02504=1174.017,4.022,-45.917,-179.997,5.903,149.053
C02505=1174.012,4.271,-45.929,-179.994,5.903,149.052
C02506=1174.007,4.521,-45.944,-179.992,5.904,149.051
C02507=1174.002,4.770,-45.958,-179.990,5.905,149.051
C02508=1173.996,5.020,-45.971,-179.987,5.905,149.050
C02509=1173.992,5.270,-45.985,-179.984,5.906,149.049
C02510=1173.987,5.519,-45.999,-179.982,5.906,149.049
C02511=1173.982,5.768,-46.013,-179.979,5.907,149.048
C02512=1173.976,6.019,-46.027,-179.977,5.908,149.048
C02513=1173.972,6.267,-46.040,-179.975,5.908,149.047
C02514=1173.967,6.517,-46.054,-179.972,5.909,149.046
C02515=1173.961,6.767,-46.068,-179.970,5.910,149.046
C02516=1173.956,7.016,-46.082,-179.967,5.910,149.045
C02517=1173.951,7.266,-46.096,-179.964,5.911,149.045
C02518=1173.947,7.515,-46.110,-179.962,5.911,149.044
C02519=1173.941,7.764,-46.123,-179.960,5.912,149.043
C02520=1173.936,8.015,-46.137,-179.957,5.912,149.043
C02521=1173.931,8.265,-46.151,-179.955,5.913,149.042
C02522=1173.925,8.514,-46.165,-179.952,5.914,149.042
C02523=1173.920,8.763,-46.179,-179.949,5.915,149.041
C02524=1173.916,9.013,-46.193,-179.947,5.916,149.041
C02525=1173.910,9.262,-46.206,-179.944,5.916,149.040
C02526=1173.905,9.512,-46.221,-179.942,5.917,149.039
C02527=1173.900,9.762,-46.235,-179.939,5.918,149.039
C02528=1173.895,10.011,-46.249,-179.937,5.918,149.038
C02529=1173.890,10.260,-46.263,-179.934,5.919,149.038
C02530=1173.885,10.510,-46.277,-179.932,5.919,149.037
C02531=1173.880,10.760,-46.290,-179.929,5.920,149.036
C02532=1173.875,11.009,-46.304,-179.927,5.921,149.036
C02533=1173.870,11.259,-46.319,-179.924,5.921,149.035
C02534=1173.865,11.509,-46.333,-179.922,5.922,149.035
C02535=1173.859,11.758,-46.347,-179.920,5.922,149.034
C02536=1173.854,12.007,-46.361,-179.916,5.924,149.033
C02537=1173.849,12.257,-46.375,-179.914,5.925,149.033
C02538=1173.845,12.507,-46.390,-179.911,5.925,149.032
C02539=1173.839,12.756,-46.403,-179.909,5.925,149.031
C02540=1173.834,13.005,-46.418,-179.907,5.926,149.031
C02541=1173.829,13.255,-46.432,-179.904,5.927,149.030
C02542=1173.824,13.505,-46.446,-179.902,5.928,149.030
C02543=1173.819,13.754,-46.460,-179.899,5.928,149.029
C02544=1173.814,14.004,-46.474,-179.897,5.929,149.028
C02545=1173.809,14.253,-46.489,-179.894,5.929,149.028
C02546=1173.804,14.503,-46.503,-179.892,5.930,149.027
C02547=1173.799,14.753,-46.517,-179.888,5.931,149.027
C02548=1173.793,15.002,-46.531,-179.886,5.932,149.026
C02549=1173.788,15.251,-46.546,-179.884,5.932,149.025
C02550=1173.783,15.501,-46.560,-179.882,5.933,149.025
C02551=1173.778,15.751,-46.574,-179.879,5.934,149.024
C02552=1173.773,16.001,-46.588,-179.876,5.934,149.024
C02553=1173.768,16.250,-46.602,-179.874,5.935,149.023
C02554=1173.763,16.499,-46.617,-179.871,5.936,149.022
C02555=1173.758,16.749,-46.631,-179.869,5.936,149.022
C02556=1173.753,16.999,-46.645,-179.867,5.937,149.021
C02557=1173.748,17.248,-46.659,-179.863,5.938,149.021
C02558=1173.742,17.497,-46.673,-179.861,5.939,149.020
C02559=1173.738,17.746,-46.688,-179.859,5.940,149.020
C02560=1173.733,17.996,-46.703,-179.856,5.940,149.019
C02561=1173.728,18.246,-46.717,-179.854,5.941,149.018
C02562=1173.723,18.496,-46.731,-179.851,5.941,149.018
C02563=1173.718,18.745,-46.745,-179.848,5.942,149.017
C02564=1173.712,18.994,-46.759,-179.846,5.943,149.017
C02565=1173.707,19.244,-46.774,-179.843,5.944,149.016
C02566=1173.703,19.493,-46.789,-179.841,5.945,149.015
C02567=1173.697,19.743,-46.803,-179.838,5.945,149.015
C02568=1173.692,19.993,-46.818,-179.836,5.946,149.014
C02569=1173.687,20.243,-46.832,-179.833,5.947,149.014
C02570=1173.682,20.492,-46.846,-179.831,5.947,149.013
C02571=1173.678,20.741,-46.861,-179.828,5.948,149.012
C02572=1173.672,20.990,-46.875,-179.826,5.948,149.012
C02573=1173.667,21.240,-46.889,-179.823,5.950,149.011
C02574=1173.662,21.490,-46.904,-179.821,5.951,149.011
C02575=1173.657,21.739,-46.919,-179.818,5.951,149.010
C02576=1173.652,21.989,-46.934,-179.815,5.952,149.009
C02577=1173.647,22.239,-46.948,-179.813,5.952,149.009
C02578=1173.642,22.488,-46.962,-179.810,5.953,149.008
C02579=1173.637,22.737,-46.977,-179.808,5.954,149.008
C02580=1173.632,22.987,-46.991,-179.805,5.955,149.007
C02581=1173.627,23.237,-47.006,-179.802,5.955,149.006
C02582=1173.621,23.486,-47.021,-179.800,5.956,149.006
C02583=1173.616,23.735,-47.035,-179.798,5.957,149.005
C02584=1173.611,23.985,-47.049,-179.795,5.957,149.005
C02585=1173.607,24.234,-47.064,-179.793,5.958,149.004
C02586=1173.601,24.484,-47.079,-179.790,5.959,149.003
C02587=1173.596,24.734,-47.094,-179.787,5.960,149.003
C02588=1173.591,24.983,-47.109,-179.785,5.961,149.002
C02589=1173.587,25.233,-47.123,-179.782,5.961,149.002
C02590=1173.581,25.483,-47.138,-179.780,5.962,149.001
C02591=1173.576,25.732,-47.153,-179.777,5.963,149.000
C02592=1173.571,25.981,-47.167,-179.775,5.963,149.000
C02593=1173.567,26.231,-47.182,-179.772,5.965,148.999
C02594=1173.561,26.481,-47.197,-179.769,5.965,148.999
C02595=1173.556,26.730,-47.212,-179.767,5.966,148.998
C02596=1173.551,26.979,-47.226,-179.764,5.967,148.998
C02597=1173.546,27.229,-47.241,-179.762,5.967,148.997
C02598=1173.541,27.478,-47.256,-179.760,5.968,148.996
C02599=1173.536,27.728,-47.270,-179.756,5.969,148.996
C02600=1173.530,27.997,-47.287,-179.754,5.970,148.995
C02601=1173.525,28.266,-47.302,-179.752,5.971,148.995
C02602=1173.520,28.535,-47.318,-179.748,5.972,148.994
C02603=1173.514,28.803,-47.335,-179.746,5.972,148.993
C02604=1173.509,29.053,-47.349,-179.744,5.973,148.993
C02605=1173.505,29.302,-47.364,-179.741,5.974,148.992
C02606=1173.499,29.552,-47.379,-179.738,5.975,148.991
C02607=1173.494,29.801,-47.394,-179.735,5.976,148.991
C02608=1173.489,30.051,-47.409,-179.733,5.976,148.990
C02609=1173.484,30.300,-47.424,-179.731,5.977,148.990
C02610=1173.479,30.550,-47.438,-179.728,5.978,148.989
C02611=1173.474,30.799,-47.454,-179.725,5.978,148.989
C02612=1173.469,31.049,-47.468,-179.723,5.980,148.988
C02613=1173.464,31.298,-47.483,-179.720,5.980,148.987
C02614=1173.459,31.548,-47.499,-179.718,5.981,148.987
C02615=1173.454,31.797,-47.513,-179.715,5.982,148.986
C02616=1173.448,32.047,-47.529,-179.713,5.982,148.986
C02617=1173.443,32.297,-47.543,-179.710,5.984,148.985
C02618=1173.439,32.546,-47.558,-179.707,5.984,148.984
C02619=1173.433,32.795,-47.573,-179.705,5.985,148.984
C02620=1173.428,33.045,-47.588,-179.702,5.986,148.983
C02621=1173.423,33.294,-47.603,-179.700,5.986,148.983
C02622=1173.419,33.544,-47.619,-179.697,5.988,148.982
C02623=1173.413,33.794,-47.634,-179.694,5.988,148.982
C02624=1173.409,34.043,-47.649,-179.692,5.989,148.981
C02625=1173.403,34.292,-47.664,-179.690,5.990,148.980
C02626=1173.398,34.542,-47.678,-179.686,5.991,148.980
C02627=1173.394,34.791,-47.693,-179.684,5.992,148.979
C02628=1173.388,35.041,-47.709,-179.681,5.992,148.979
C02629=1173.384,35.290,-47.724,-179.679,5.993,148.978
C02630=1173.378,35.540,-47.739,-179.677,5.994,148.977
C02631=1173.374,35.790,-47.754,-179.673,5.995,148.977
C02632=1173.368,36.039,-47.770,-179.671,5.996,148.976
C02633=1173.363,36.288,-47.785,-179.669,5.996,148.976
C02634=1173.358,36.538,-47.800,-179.666,5.997,148.975
C02635=1173.353,36.787,-47.815,-179.664,5.998,148.975
C02636=1173.348,37.037,-47.830,-179.661,5.999,148.974
C02637=1173.343,37.286,-47.846,-179.658,6.000,148.973
C02638=1173.338,37.535,-47.861,-179.656,6.000,148.973
C02639=1173.333,37.786,-47.876,-179.654,6.001,148.972
C02640=1173.328,38.035,-47.891,-179.650,6.002,148.972
C02641=1173.323,38.284,-47.907,-179.648,6.003,148.971
C02642=1173.318,38.533,-47.922,-179.646,6.004,148.971
C02643=1173.313,38.783,-47.937,-179.643,6.004,148.970
C02644=1173.307,39.032,-47.953,-179.640,6.006,148.969
C02645=1173.303,39.282,-47.968,-179.638,6.006,148.969
C02646=1173.298,39.532,-47.983,-179.635,6.007,148.968
C02647=1173.293,39.781,-47.998,-179.633,6.008,148.968
C02648=1173.288,40.030,-48.014,-179.630,6.009,148.967
C02649=1173.282,40.280,-48.029,-179.627,6.010,148.966
C02650=1173.278,40.530,-48.045,-179.625,6.010,148.966
C02651=1173.273,40.779,-48.060,-179.623,6.011,148.965
C02652=1173.268,41.028,-48.076,-179.619,6.013,148.965
C02653=1173.263,41.278,-48.091,-179.617,6.013,148.964
C02654=1173.257,41.527,-48.106,-179.615,6.014,148.964
C02655=1173.253,41.777,-48.122,-179.612,6.015,148.963
C02656=1173.248,42.026,-48.137,-179.609,6.016,148.962
C02657=1173.243,42.276,-48.153,-179.607,6.017,148.962
C02658=1173.237,42.525,-48.168,-179.604,6.018,148.961
C02659=1173.233,42.775,-48.184,-179.602,6.018,148.961
C02660=1173.228,43.024,-48.199,-179.599,6.020,148.960
C02661=1173.222,43.274,-48.215,-179.596,6.020,148.960
C02662=1173.218,43.523,-48.230,-179.594,6.021,148.959
C02663=1173.213,43.773,-48.246,-179.592,6.022,148.958
C02664=1173.208,44.022,-48.262,-179.588,6.023,148.958
C02665=1173.203,44.271,-48.277,-179.586,6.024,148.957
C02666=1173.198,44.521,-48.292,-179.584,6.024,148.957
C02667=1173.193,44.771,-48.308,-179.581,6.026,148.956
C02668=1173.187,45.020,-48.324,-179.578,6.026,148.956
C02669=1173.183,45.269,-48.339,-179.576,6.027,148.955
C02670=1173.177,45.519,-48.354,-179.573,6.028,148.954
C02671=1173.173,45.769,-48.370,-179.571,6.029,148.954
C02672=1173.168,46.018,-48.386,-179.568,6.030,148.953
C02673=1173.163,46.267,-48.401,-179.565,6.030,148.953
C02674=1173.158,46.517,-48.417,-179.563,6.031,148.952
C02675=1173.153,46.766,-48.433,-179.560,6.033,148.952
C02676=1173.147,47.016,-48.449,-179.558,6.033,148.951
C02677=1173.143,47.265,-48.464,-179.555,6.034,148.950
C02678=1173.138,47.515,-48.480,-179.552,6.036,148.950
C02679=1173.133,47.763,-48.496,-179.550,6.036,148.949
C02680=1173.128,48.014,-48.512,-179.548,6.037,148.949
C02681=1173.123,48.263,-48.527,-179.544,6.038,148.948
C02682=1173.117,48.512,-48.543,-179.542,6.039,148.948
C02683=1173.113,48.762,-48.558,-179.540,6.040,148.947
C02684=1173.108,49.011,-48.575,-179.537,6.040,148.946
C02685=1173.103,49.260,-48.590,-179.534,6.042,148.946
C02686=1173.098,49.510,-48.606,-179.532,6.042,148.945
C02687=1173.093,49.760,-48.622,-179.529,6.043,148.945
C02688=1173.087,50.009,-48.638,-179.526,6.045,148.944
C02689=1173.083,50.258,-48.653,-179.524,6.045,148.944
C02690=1173.078,50.508,-48.669,-179.521,6.046,148.943
C02691=1173.074,50.757,-48.686,-179.519,6.048,148.943
C02692=1173.068,51.007,-48.701,-179.516,6.048,148.942
C02693=1173.063,51.256,-48.717,-179.513,6.049,148.941
C02694=1173.058,51.506,-48.733,-179.511,6.050,148.941
C02695=1173.053,51.755,-48.749,-179.508,6.051,148.940
C02696=1173.048,52.004,-48.765,-179.506,6.052,148.940
C02697=1173.043,52.254,-48.781,-179.503,6.052,148.939
C02698=1173.038,52.503,-48.796,-179.501,6.054,148.939
C02699=1173.034,52.753,-48.812,-179.498,6.054,148.938
C02700=1173.029,53.002,-48.829,-179.496,6.055,148.938
C02701=1173.023,53.251,-48.844,-179.492,6.057,148.937
C02702=1173.018,53.501,-48.860,-179.490,6.057,148.936
C02703=1173.013,53.750,-48.876,-179.488,6.058,148.936
C02704=1173.008,54.019,-48.894,-179.484,6.059,148.935
C02705=1173.003,54.288,-48.911,-179.482,6.060,148.935
C02706=1172.997,54.556,-48.928,-179.479,6.061,148.934
C02707=1172.992,54.824,-48.946,-179.476,6.062,148.933
C02708=1172.987,55.074,-48.962,-179.474,6.064,148.933
C02709=1172.982,55.324,-48.977,-179.471,6.064,148.932
C02710=1172.977,55.573,-48.994,-179.469,6.065,148.932
C02711=1172.972,55.823,-49.009,-179.466,6.066,148.931
C02712=1172.967,56.072,-49.026,-179.463,6.067,148.930
C02713=1172.962,56.321,-49.042,-179.460,6.069,148.930
C02714=1172.958,56.571,-49.058,-179.458,6.069,148.929
C02715=1172.951,56.821,-49.075,-179.456,6.070,148.929
C02716=1172.947,57.070,-49.091,-179.452,6.071,148.928
C02717=1172.942,57.320,-49.107,-179.450,6.072,148.928
C02718=1172.936,57.568,-49.123,-179.448,6.073,148.927
C02719=1172.932,57.818,-49.140,-179.445,6.074,148.927
C02720=1172.927,58.067,-49.155,-179.442,6.075,148.926
C02721=1172.922,58.317,-49.172,-179.440,6.076,148.926
C02722=1172.917,58.566,-49.188,-179.437,6.077,148.925
C02723=1172.912,58.816,-49.204,-179.435,6.078,148.925
C02724=1172.907,59.065,-49.220,-179.432,6.078,148.924
C02725=1172.902,59.314,-49.237,-179.429,6.080,148.923
C02726=1172.898,59.564,-49.253,-179.427,6.081,148.923
C02727=1172.893,59.813,-49.269,-179.424,6.082,148.922
C02728=1172.887,60.063,-49.286,-179.421,6.083,148.922
C02729=1172.882,60.312,-49.302,-179.419,6.084,148.921
C02730=1172.877,60.562,-49.318,-179.416,6.085,148.921
C02731=1172.872,60.811,-49.335,-179.414,6.086,148.920
C02732=1172.868,61.060,-49.351,-179.411,6.086,148.919
C02733=1172.863,61.310,-49.367,-179.408,6.088,148.919
C02734=1172.858,61.559,-49.384,-179.406,6.089,148.918
C02735=1172.852,61.808,-49.400,-179.404,6.089,148.918
C02736=1172.847,62.058,-49.416,-179.400,6.091,148.917
C02737=1172.843,62.308,-49.433,-179.398,6.092,148.917
C02738=1172.838,62.557,-49.449,-179.395,6.093,148.916
C02739=1172.833,62.806,-49.466,-179.393,6.094,148.916
C02740=1172.827,63.056,-49.482,-179.390,6.094,148.915
C02741=1172.823,63.305,-49.499,-179.387,6.096,148.915
C02742=1172.818,63.554,-49.515,-179.385,6.097,148.914
C02743=1172.813,63.804,-49.532,-179.382,6.098,148.914
C02744=1172.808,64.054,-49.548,-179.379,6.099,148.913
C02745=1172.803,64.303,-49.565,-179.377,6.100,148.912
C02746=1172.798,64.552,-49.581,-179.374,6.101,148.912
C02747=1172.794,64.802,-49.598,-179.372,6.102,148.911
C02748=1172.789,65.051,-49.614,-179.369,6.103,148.911
C02749=1172.783,65.300,-49.632,-179.367,6.104,148.910
C02750=1172.778,65.550,-49.647,-179.364,6.105,148.910
C02751=1172.773,65.799,-49.664,-179.361,6.106,148.909
C02752=1172.769,66.049,-49.681,-179.359,6.107,148.908
C02753=1172.763,66.298,-49.697,-179.356,6.108,148.908
C02754=1172.759,66.547,-49.714,-179.353,6.109,148.907
C02755=1172.754,66.797,-49.731,-179.351,6.110,148.907
C02756=1172.748,67.046,-49.748,-179.348,6.111,148.906
C02757=1172.744,67.295,-49.764,-179.346,6.112,148.906
C02758=1172.739,67.545,-49.780,-179.343,6.113,148.905
C02759=1172.733,67.795,-49.797,-179.340,6.114,148.905
C02760=1172.729,68.044,-49.814,-179.337,6.116,148.904
C02761=1172.724,68.294,-49.831,-179.335,6.116,148.904
C02762=1172.719,68.543,-49.847,-179.332,6.117,148.903
C02763=1172.714,68.792,-49.864,-179.330,6.119,148.903
C02764=1172.710,69.042,-49.881,-179.327,6.119,148.902
C02765=1172.704,69.291,-49.898,-179.324,6.121,148.902
C02766=1172.699,69.540,-49.914,-179.322,6.121,148.901
C02767=1172.695,69.790,-49.931,-179.320,6.122,148.900
C02768=1172.689,70.039,-49.948,-179.316,6.124,148.900
C02769=1172.685,70.288,-49.965,-179.314,6.125,148.899
C02770=1172.680,70.538,-49.981,-179.311,6.126,148.899
C02771=1172.675,70.788,-49.999,-179.309,6.127,148.898
C02772=1172.670,71.036,-50.015,-179.306,6.128,148.898
C02773=1172.665,71.286,-50.032,-179.303,6.129,148.897
C02774=1172.660,71.536,-50.049,-179.301,6.131,148.897
C02775=1172.655,71.784,-50.066,-179.298,6.131,148.896
C02776=1172.650,72.034,-50.083,-179.296,6.132,148.896
C02777=1172.646,72.283,-50.100,-179.293,6.133,148.895
C02778=1172.640,72.533,-50.117,-179.291,6.134,148.895
C02779=1172.635,72.782,-50.133,-179.287,6.136,148.894
C02780=1172.630,73.031,-50.151,-179.285,6.136,148.893
C02781=1172.626,73.281,-50.167,-179.282,6.138,148.893
C02782=1172.620,73.531,-50.184,-179.280,6.139,148.892
C02783=1172.616,73.779,-50.202,-179.277,6.140,148.892
C02784=1172.610,74.029,-50.219,-179.274,6.141,148.891
C02785=1172.606,74.278,-50.235,-179.271,6.142,148.891
C02786=1172.601,74.528,-50.253,-179.269,6.143,148.890
C02787=1172.596,74.777,-50.269,-179.266,6.144,148.890
C02788=1172.590,75.026,-50.286,-179.264,6.145,148.889
C02789=1172.586,75.275,-50.304,-179.262,6.146,148.889
C02790=1172.581,75.525,-50.321,-179.258,6.148,148.888
C02791=1172.576,75.775,-50.338,-179.256,6.148,148.888
C02792=1172.571,76.024,-50.355,-179.253,6.150,148.887
C02793=1172.566,76.273,-50.372,-179.251,6.151,148.887
C02794=1172.561,76.522,-50.389,-179.248,6.152,148.886
C02795=1172.556,76.772,-50.406,-179.246,6.153,148.885
C02796=1172.552,77.022,-50.423,-179.242,6.154,148.885
C02797=1172.547,77.271,-50.441,-179.240,6.155,148.884
C02798=1172.542,77.520,-50.458,-179.237,6.157,148.884
C02799=1172.536,77.769,-50.475,-179.235,6.157,148.883
C02800=1172.532,78.018,-50.492,-179.232,6.159,148.883
C02801=1172.527,78.268,-50.509,-179.229,6.160,148.882
C02802=1172.522,78.518,-50.527,-179.227,6.161,148.882
C02803=1172.518,78.767,-50.544,-179.224,6.162,148.881
C02804=1172.512,79.017,-50.561,-179.221,6.163,148.881
C02805=1172.507,79.266,-50.578,-179.219,6.164,148.880
C02806=1172.502,79.514,-50.595,-179.216,6.166,148.880
C02807=1172.497,79.764,-50.613,-179.214,6.167,148.879
C02808=1172.492,80.033,-50.632,-179.211,6.168,148.879
C02809=1172.487,80.301,-50.650,-179.208,6.168,148.878
C02810=1172.481,80.569,-50.669,-179.205,6.170,148.877
C02811=1172.476,80.838,-50.687,-179.202,6.172,148.877
C02812=1172.472,81.087,-50.705,-179.200,6.172,148.876
C02813=1172.467,81.337,-50.722,-179.197,6.174,148.876
C02814=1172.462,81.586,-50.740,-179.195,6.175,148.875
C02815=1172.457,81.836,-50.757,-179.191,6.176,148.875
C02816=1172.452,82.085,-50.775,-179.189,6.177,148.874
C02817=1172.447,82.334,-50.791,-179.187,6.179,148.874
C02818=1172.442,82.583,-50.809,-179.184,6.179,148.873
C02819=1172.437,82.832,-50.826,-179.181,6.181,148.873
C02820=1172.432,83.082,-50.844,-179.179,6.181,148.872
C02821=1172.427,83.331,-50.861,-179.176,6.183,148.872
C02822=1172.422,83.581,-50.879,-179.173,6.184,148.871
C02823=1172.418,83.830,-50.896,-179.170,6.185,148.871
C02824=1172.413,84.079,-50.914,-179.168,6.186,148.870
C02825=1172.407,84.329,-50.931,-179.165,6.187,148.870
C02826=1172.403,84.578,-50.949,-179.163,6.188,148.869
C02827=1172.398,84.827,-50.967,-179.160,6.190,148.868
C02828=1172.393,85.077,-50.984,-179.157,6.191,148.868
C02829=1172.388,85.326,-51.002,-179.154,6.192,148.867
C02830=1172.383,85.576,-51.019,-179.152,6.194,148.867
C02831=1172.378,85.825,-51.037,-179.150,6.195,148.867
C02832=1172.374,86.074,-51.054,-179.146,6.196,148.866
C02833=1172.369,86.324,-51.072,-179.144,6.197,148.865
C02834=1172.364,86.573,-51.090,-179.141,6.198,148.865
C02835=1172.359,86.822,-51.108,-179.139,6.199,148.864
C02836=1172.354,87.072,-51.125,-179.136,6.201,148.864
C02837=1172.349,87.321,-51.143,-179.134,6.201,148.863
C02838=1172.344,87.570,-51.161,-179.131,6.203,148.863
C02839=1172.339,87.820,-51.178,-179.128,6.204,148.862
C02840=1172.334,88.069,-51.196,-179.125,6.205,148.862
C02841=1172.330,88.318,-51.214,-179.123,6.207,148.861
C02842=1172.325,88.567,-51.232,-179.120,6.207,148.861
C02843=1172.319,88.817,-51.249,-179.117,6.209,148.860
C02844=1172.315,89.066,-51.267,-179.115,6.210,148.860
C02845=1172.310,89.315,-51.285,-179.112,6.211,148.859
C02846=1172.305,89.564,-51.303,-179.110,6.212,148.859
C02847=1172.299,89.814,-51.320,-179.107,6.214,148.858
C02848=1172.295,90.063,-51.337,-179.105,6.215,148.858
C02849=1172.290,90.312,-51.355,-179.101,6.216,148.857
C02850=1172.285,90.561,-51.373,-179.099,6.218,148.857
C02851=1172.281,90.811,-51.391,-179.096,6.218,148.856
C02852=1172.276,91.060,-51.409,-179.093,6.220,148.856
C02853=1172.270,91.310,-51.427,-179.091,6.221,148.855
C02854=1172.266,91.560,-51.445,-179.088,6.222,148.855
C02855=1172.261,91.809,-51.463,-179.086,6.223,148.854
C02856=1172.256,92.058,-51.481,-179.083,6.225,148.854
C02857=1172.251,92.307,-51.499,-179.080,6.226,148.853
C02858=1172.246,92.556,-51.517,-179.078,6.227,148.853
C02859=1172.242,92.805,-51.535,-179.075,6.229,148.852
C02860=1172.237,93.055,-51.553,-179.072,6.229,148.852
C02861=1172.231,93.304,-51.570,-179.070,6.231,148.851
C02862=1172.227,93.554,-51.588,-179.067,6.233,148.851
C02863=1172.222,93.803,-51.606,-179.064,6.233,148.850
C02864=1172.217,94.053,-51.624,-179.062,6.235,148.850
C02865=1172.212,94.302,-51.642,-179.059,6.235,148.849
C02866=1172.207,94.551,-51.660,-179.056,6.237,148.849
C02867=1172.203,94.800,-51.678,-179.054,6.238,148.848
C02868=1172.198,95.049,-51.696,-179.051,6.239,148.848
C02869=1172.193,95.298,-51.714,-179.048,6.241,148.847
C02870=1172.188,95.548,-51.732,-179.046,6.242,148.847
C02871=1172.183,95.798,-51.751,-179.043,6.243,148.846
C02872=1172.178,96.047,-51.769,-179.041,6.244,148.846
C02873=1172.173,96.296,-51.787,-179.038,6.246,148.845
C02874=1172.168,96.545,-51.805,-179.035,6.247,148.845
C02875=1172.163,96.795,-51.823,-179.033,6.248,148.844
C02876=1172.159,97.043,-51.842,-179.029,6.250,148.844
C02877=1172.154,97.293,-51.860,-179.027,6.251,148.843
C02878=1172.149,97.542,-51.878,-179.025,6.252,148.843
C02879=1172.144,97.791,-51.896,-179.021,6.253,148.842
C02880=1172.139,98.041,-51.915,-179.019,6.254,148.842
C02881=1172.134,98.290,-51.933,-179.017,6.256,148.841
C02882=1172.130,98.540,-51.951,-179.013,6.257,148.841
C02883=1172.125,98.789,-51.969,-179.011,6.258,148.840
C02884=1172.120,99.038,-51.987,-179.008,6.260,148.840
C02885=1172.115,99.287,-52.006,-179.006,6.261,148.839
C02886=1172.109,99.536,-52.024,-179.003,6.262,148.839
C02887=1172.105,99.786,-52.043,-179.000,6.264,148.838
C02888=1172.100,100.035,-52.061,-178.998,6.265,148.838
C02889=1172.095,100.284,-52.079,-178.995,6.266,148.837
C02890=1172.091,100.533,-52.097,-178.992,6.268,148.837
C02891=1172.086,100.783,-52.116,-178.990,6.269,148.836
C02892=1172.081,101.032,-52.134,-178.987,6.270,148.836
C02893=1172.076,101.282,-52.152,-178.984,6.272,148.835
C02894=1172.071,101.530,-52.171,-178.982,6.273,148.835
C02895=1172.066,101.780,-52.190,-178.979,6.274,148.834
C02896=1172.061,102.029,-52.208,-178.977,6.275,148.834
C02897=1172.056,102.279,-52.226,-178.974,6.277,148.833
C02898=1172.052,102.527,-52.244,-178.971,6.278,148.833
C02899=1172.047,102.777,-52.263,-178.969,6.279,148.832
C02900=1172.042,103.027,-52.281,-178.966,6.280,148.832
C02901=1172.037,103.275,-52.300,-178.963,6.282,148.831
C02902=1172.033,103.525,-52.318,-178.961,6.283,148.831
C02903=1172.027,103.775,-52.337,-178.958,6.284,148.830
C02904=1172.023,104.023,-52.356,-178.955,6.286,148.830
C02905=1172.018,104.273,-52.374,-178.953,6.287,148.830
C02906=1172.013,104.522,-52.393,-178.950,6.288,148.829
C02907=1172.008,104.771,-52.411,-178.947,6.290,148.828
C02908=1172.004,105.021,-52.430,-178.945,6.291,148.828
C02909=1171.998,105.270,-52.449,-178.941,6.292,148.827
C02910=1171.993,105.519,-52.467,-178.939,6.294,148.827
C02911=1171.989,105.768,-52.485,-178.937,6.295,148.827
C02912=1171.984,106.037,-52.506,-178.933,6.296,148.826
C02913=1171.978,106.305,-52.526,-178.931,6.298,148.826
C02914=1171.973,106.574,-52.545,-178.927,6.300,148.825
C02915=1171.968,106.842,-52.566,-178.925,6.301,148.825
C02916=1171.963,107.091,-52.584,-178.923,6.302,148.824
C02917=1171.958,107.340,-52.603,-178.919,6.303,148.823
C02918=1171.953,107.590,-52.622,-178.917,6.305,148.823
C02919=1171.949,107.839,-52.641,-178.914,6.307,148.823
C02920=1171.943,108.088,-52.659,-178.911,6.307,148.822
C02921=1171.939,108.337,-52.678,-178.909,6.309,148.822
C02922=1171.933,108.587,-52.697,-178.906,6.311,148.821
C02923=1171.929,108.836,-52.716,-178.903,6.311,148.821
C02924=1171.925,109.085,-52.735,-178.901,6.313,148.820
C02925=1171.919,109.334,-52.753,-178.898,6.315,148.820
C02926=1171.915,109.583,-52.772,-178.896,6.316,148.819
C02927=1171.909,109.833,-52.791,-178.893,6.317,148.819
C02928=1171.905,110.082,-52.810,-178.890,6.319,148.818
C02929=1171.900,110.332,-52.829,-178.888,6.320,148.818
C02930=1171.895,110.580,-52.847,-178.885,6.321,148.817
C02931=1171.890,110.830,-52.867,-178.882,6.323,148.817
C02932=1171.886,111.079,-52.885,-178.879,6.325,148.816
C02933=1171.881,111.329,-52.905,-178.877,6.326,148.816
C02934=1171.876,111.577,-52.923,-178.874,6.327,148.815
C02935=1171.871,111.827,-52.942,-178.871,6.329,148.815
C02936=1171.867,112.076,-52.961,-178.869,6.330,148.815
C02937=1171.862,112.325,-52.981,-178.866,6.331,148.814
C02938=1171.856,112.575,-52.999,-178.863,6.333,148.814
C02939=1171.852,112.823,-53.018,-178.860,6.334,148.813
C02940=1171.847,113.073,-53.037,-178.858,6.335,148.813
C02941=1171.842,113.322,-53.056,-178.855,6.337,148.812
C02942=1171.837,113.572,-53.075,-178.852,6.338,148.812
C02943=1171.833,113.820,-53.094,-178.850,6.339,148.811
C02944=1171.828,114.070,-53.113,-178.847,6.341,148.811
C02945=1171.822,114.319,-53.133,-178.844,6.342,148.810
C02946=1171.818,114.569,-53.151,-178.842,6.344,148.810
C02947=1171.813,114.818,-53.170,-178.839,6.345,148.809
C02948=1171.809,115.067,-53.189,-178.836,6.346,148.809
C02949=1171.803,115.316,-53.209,-178.834,6.348,148.808
C02950=1171.799,115.565,-53.228,-178.831,6.349,148.808
C02951=1171.794,115.814,-53.247,-178.829,6.351,148.808
C02952=1171.789,116.064,-53.266,-178.825,6.352,148.807
C02953=1171.784,116.313,-53.285,-178.823,6.354,148.807
C02954=1171.780,116.562,-53.304,-178.821,6.355,148.806
C02955=1171.774,116.811,-53.324,-178.818,6.356,148.806
C02956=1171.770,117.061,-53.343,-178.815,6.358,148.805
C02957=1171.766,117.310,-53.362,-178.812,6.360,148.805
C02958=1171.760,117.559,-53.382,-178.810,6.360,148.804
C02959=1171.755,117.808,-53.401,-178.807,6.362,148.804
C02960=1171.750,118.057,-53.421,-178.804,6.364,148.803
C02961=1171.746,118.306,-53.440,-178.801,6.365,148.803
C02962=1171.741,118.556,-53.458,-178.799,6.366,148.802
C02963=1171.736,118.805,-53.478,-178.796,6.368,148.802
C02964=1171.732,119.055,-53.497,-178.794,6.370,148.802
C02965=1171.726,119.304,-53.516,-178.791,6.371,148.801
C02966=1171.722,119.553,-53.536,-178.788,6.372,148.801
C02967=1171.716,119.802,-53.555,-178.786,6.374,148.800
C02968=1171.712,120.051,-53.574,-178.783,6.375,148.800
C02969=1171.707,120.300,-53.594,-178.780,6.377,148.799
C02970=1171.702,120.550,-53.613,-178.777,6.378,148.799
C02971=1171.698,120.799,-53.634,-178.775,6.379,148.798
C02972=1171.692,121.047,-53.653,-178.772,6.381,148.798
C02973=1171.688,121.297,-53.672,-178.769,6.383,148.797
C02974=1171.684,121.546,-53.692,-178.766,6.384,148.797
C02975=1171.678,121.795,-53.711,-178.764,6.385,148.797
C02976=1171.674,122.045,-53.731,-178.762,6.387,148.796
C02977=1171.668,122.294,-53.750,-178.759,6.389,148.796
C02978=1171.664,122.543,-53.769,-178.756,6.390,148.795
C02979=1171.660,122.792,-53.789,-178.753,6.392,148.795
C02980=1171.654,123.041,-53.808,-178.751,6.393,148.794
C02981=1171.650,123.290,-53.828,-178.748,6.394,148.794
C02982=1171.645,123.540,-53.848,-178.745,6.396,148.793
C02983=1171.640,123.789,-53.867,-178.742,6.397,148.793
C02984=1171.635,124.038,-53.887,-178.740,6.398,148.793
C02985=1171.631,124.287,-53.906,-178.737,6.400,148.792
C02986=1171.626,124.536,-53.926,-178.735,6.402,148.792
C02987=1171.621,124.785,-53.946,-178.731,6.403,148.791
C02988=1171.616,125.035,-53.965,-178.729,6.405,148.791
C02989=1171.612,125.284,-53.985,-178.727,6.406,148.790
C02990=1171.606,125.533,-54.004,-178.724,6.408,148.790
C02991=1171.602,125.782,-54.025,-178.721,6.409,148.790
C02992=1171.597,126.032,-54.044,-178.718,6.411,148.789
C02993=1171.592,126.281,-54.063,-178.715,6.412,148.789
C02994=1171.587,126.530,-54.084,-178.713,6.414,148.788
C02995=1171.583,126.779,-54.103,-178.711,6.415,148.788
C02996=1171.578,127.029,-54.123,-178.708,6.417,148.787
C02997=1171.573,127.278,-54.142,-178.705,6.418,148.787
C02998=1171.568,127.527,-54.163,-178.702,6.420,148.786
C02999=1171.563,127.776,-54.182,-178.699,6.422,148.786
C03000=1171.560,128.025,-54.202,-178.697,6.423,148.785
C03001=1171.554,128.274,-54.222,-178.694,6.424,148.785
C03002=1171.550,128.523,-54.241,-178.692,6.426,148.785
C03003=1171.545,128.772,-54.262,-178.688,6.427,148.784
C03004=1171.540,129.022,-54.282,-178.686,6.429,148.784
C03005=1171.534,129.271,-54.301,-178.683,6.431,148.783
C03006=1171.530,129.520,-54.321,-178.681,6.432,148.783
C03007=1171.525,129.769,-54.341,-178.678,6.434,148.782
C03008=1171.521,130.018,-54.362,-178.676,6.435,148.782
C03009=1171.515,130.267,-54.381,-178.672,6.437,148.781
C03010=1171.511,130.516,-54.401,-178.670,6.438,148.781
C03011=1171.506,130.766,-54.421,-178.667,6.440,148.781
C03012=1171.502,131.015,-54.441,-178.665,6.441,148.780
C03013=1171.497,131.264,-54.461,-178.662,6.443,148.780
C03014=1171.492,131.513,-54.481,-178.659,6.445,148.780
C03015=1171.487,131.762,-54.501,-178.656,6.446,148.779
C03016=1171.482,132.031,-54.522,-178.654,6.448,148.779
C03017=1171.477,132.299,-54.544,-178.651,6.449,148.778
C03018=1171.471,132.568,-54.566,-178.648,6.451,148.777
C03019=1171.466,132.837,-54.587,-178.645,6.453,148.777
C03020=1171.462,133.086,-54.607,-178.642,6.454,148.777
C03021=1171.457,133.335,-54.628,-178.640,6.456,148.776
C03022=1171.452,133.584,-54.648,-178.637,6.458,148.776
C03023=1171.448,133.833,-54.668,-178.634,6.459,148.775
C03024=1171.442,134.082,-54.687,-178.631,6.461,148.775
C03025=1171.438,134.331,-54.708,-178.629,6.462,148.775
C03026=1171.433,134.580,-54.728,-178.626,6.464,148.774
C03027=1171.428,134.830,-54.748,-178.623,6.465,148.774
C03028=1171.423,135.079,-54.769,-178.621,6.467,148.773
C03029=1171.419,135.328,-54.789,-178.618,6.469,148.773
C03030=1171.414,135.578,-54.809,-178.615,6.470,148.772
C03031=1171.410,135.826,-54.829,-178.612,6.472,148.772
C03032=1171.404,136.075,-54.850,-178.610,6.473,148.772
C03033=1171.399,136.325,-54.869,-178.607,6.475,148.771
C03034=1171.395,136.574,-54.890,-178.605,6.476,148.771
C03035=1171.390,136.823,-54.910,-178.602,6.478,148.770
C03036=1171.385,137.072,-54.931,-178.599,6.480,148.770
C03037=1171.380,137.321,-54.951,-178.597,6.481,148.770
C03038=1171.376,137.570,-54.971,-178.593,6.483,148.769
C03039=1171.372,137.819,-54.992,-178.591,6.485,148.769
C03040=1171.366,138.069,-55.013,-178.588,6.486,148.768
C03041=1171.362,138.318,-55.032,-178.586,6.487,148.768
C03042=1171.357,138.567,-55.053,-178.583,6.489,148.767
C03043=1171.352,138.816,-55.074,-178.580,6.491,148.767
C03044=1171.348,139.065,-55.094,-178.578,6.493,148.767
C03045=1171.343,139.314,-55.114,-178.575,6.494,148.766
C03046=1171.338,139.563,-55.135,-178.572,6.496,148.766
C03047=1171.333,139.812,-55.155,-178.569,6.497,148.765
C03048=1171.328,140.061,-55.175,-178.566,6.499,148.765
C03049=1171.323,140.311,-55.196,-178.564,6.501,148.765
C03050=1171.319,140.559,-55.216,-178.561,6.503,148.764
C03051=1171.314,140.808,-55.237,-178.559,6.504,148.764
C03052=1171.309,141.058,-55.258,-178.556,6.505,148.763
C03053=1171.305,141.307,-55.278,-178.554,6.507,148.763
C03054=1171.300,141.556,-55.298,-178.551,6.509,148.763
C03055=1171.295,141.805,-55.319,-178.548,6.511,148.762
C03056=1171.291,142.054,-55.340,-178.545,6.512,148.762
C03057=1171.285,142.303,-55.361,-178.542,6.514,148.761
C03058=1171.281,142.552,-55.381,-178.540,6.515,148.761
C03059=1171.276,142.801,-55.401,-178.537,6.517,148.760
C03060=1171.271,143.050,-55.422,-178.534,6.519,148.760
C03061=1171.267,143.300,-55.443,-178.531,6.521,148.760
C03062=1171.262,143.549,-55.464,-178.529,6.522,148.759
C03063=1171.258,143.798,-55.484,-178.526,6.524,148.759
C03064=1171.253,144.047,-55.505,-178.524,6.525,148.758
C03065=1171.248,144.296,-55.526,-178.521,6.527,148.758
C03066=1171.243,144.546,-55.547,-178.519,6.529,148.758
C03067=1171.239,144.794,-55.567,-178.515,6.530,148.757
C03068=1171.233,145.044,-55.588,-178.513,6.532,148.757
C03069=1171.229,145.293,-55.608,-178.510,6.533,148.756
C03070=1171.224,145.542,-55.629,-178.507,6.535,148.756
C03071=1171.219,145.791,-55.650,-178.505,6.537,148.756
C03072=1171.215,146.040,-55.671,-178.502,6.539,148.755
C03073=1171.210,146.288,-55.692,-178.499,6.540,148.755
C03074=1171.205,146.538,-55.713,-178.496,6.542,148.754
C03075=1171.201,146.787,-55.733,-178.494,6.544,148.754
C03076=1171.196,147.037,-55.754,-178.491,6.546,148.754
C03077=1171.191,147.286,-55.775,-178.488,6.547,148.753
C03078=1171.187,147.534,-55.797,-178.486,6.549,148.753
C03079=1171.182,147.783,-55.817,-178.483,6.551,148.753
C03080=1171.177,148.032,-55.838,-178.480,6.553,148.752
C03081=1171.172,148.282,-55.859,-178.478,6.554,148.752
C03082=1171.167,148.531,-55.879,-178.475,6.556,148.751
C03083=1171.163,148.779,-55.901,-178.472,6.558,148.751
C03084=1171.159,149.029,-55.922,-178.470,6.558,148.750
C03085=1171.154,149.278,-55.943,-178.467,6.560,148.750
C03086=1171.149,149.527,-55.964,-178.464,6.562,148.750
C03087=1171.144,149.776,-55.985,-178.462,6.564,148.749
C03088=1171.139,150.025,-56.006,-178.459,6.565,148.749
C03089=1171.134,150.274,-56.027,-178.456,6.567,148.748
C03090=1171.130,150.523,-56.048,-178.453,6.569,148.748
C03091=1171.125,150.773,-56.069,-178.451,6.571,148.748
C03092=1171.120,151.022,-56.090,-178.448,6.572,148.747
C03093=1171.116,151.270,-56.111,-178.445,6.574,148.747
C03094=1171.111,151.519,-56.132,-178.443,6.576,148.747
C03095=1171.106,151.768,-56.154,-178.440,6.578,148.746
C03096=1171.102,152.018,-56.174,-178.437,6.579,148.746
C03097=1171.097,152.267,-56.195,-178.435,6.581,148.745
C03098=1171.092,152.516,-56.217,-178.432,6.583,148.745
C03099=1171.087,152.765,-56.238,-178.429,6.585,148.745
C03100=1171.083,153.013,-56.259,-178.427,6.586,148.744
C03101=1171.078,153.263,-56.280,-178.424,6.588,148.744
C03102=1171.073,153.512,-56.302,-178.421,6.590,148.744
C03103=1171.068,153.761,-56.323,-178.418,6.592,148.743
C03104=1171.064,154.010,-56.344,-178.416,6.593,148.743
C03105=1171.059,154.259,-56.366,-178.413,6.595,148.742
C03106=1171.054,154.509,-56.387,-178.410,6.597,148.742
C03107=1171.049,154.757,-56.408,-178.408,6.599,148.742
C03108=1171.045,155.006,-56.429,-178.405,6.600,148.741
C03109=1171.041,155.256,-56.451,-178.402,6.602,148.741
C03110=1171.036,155.504,-56.472,-178.400,6.604,148.741
C03111=1171.031,155.753,-56.493,-178.397,6.606,148.740
C03112=1171.026,156.002,-56.515,-178.394,6.607,148.740
C03113=1171.021,156.252,-56.536,-178.392,6.609,148.739
C03114=1171.017,156.500,-56.557,-178.389,6.611,148.739
C03115=1171.012,156.749,-56.579,-178.386,6.613,148.739
C03116=1171.007,156.998,-56.600,-178.383,6.614,148.738
C03117=1171.003,157.248,-56.622,-178.381,6.616,148.738
C03118=1170.997,157.497,-56.643,-178.378,6.618,148.737
C03119=1170.993,157.746,-56.665,-178.375,6.620,148.737
C03120=1170.988,158.015,-56.687,-178.372,6.622,148.737
C03121=1170.983,158.283,-56.712,-178.369,6.624,148.736
C03122=1170.978,158.552,-56.734,-178.366,6.625,148.736
C03123=1170.972,158.822,-56.758,-178.363,6.628,148.735
C03124=1170.968,159.070,-56.779,-178.360,6.630,148.735
C03125=1170.964,159.319,-56.801,-178.358,6.632,148.735
C03126=1170.959,159.569,-56.822,-178.355,6.633,148.734
C03127=1170.954,159.817,-56.843,-178.352,6.635,148.734
C03128=1170.950,160.067,-56.866,-178.350,6.637,148.734
C03129=1170.945,160.315,-56.887,-178.347,6.639,148.733
C03130=1170.940,160.565,-56.909,-178.344,6.640,148.733
C03131=1170.935,160.814,-56.930,-178.341,6.642,148.732
C03132=1170.931,161.063,-56.952,-178.339,6.644,148.732
C03133=1170.926,161.312,-56.974,-178.337,6.646,148.732
C03134=1170.921,161.561,-56.996,-178.334,6.648,148.732
C03135=1170.916,161.810,-57.017,-178.331,6.649,148.731
C03136=1170.912,162.059,-57.039,-178.328,6.651,148.731
C03137=1170.907,162.308,-57.060,-178.326,6.653,148.730
C03138=1170.903,162.557,-57.082,-178.323,6.655,148.730
C03139=1170.898,162.806,-57.104,-178.320,6.656,148.730
C03140=1170.893,163.054,-57.126,-178.317,6.659,148.729
C03141=1170.889,163.304,-57.148,-178.314,6.661,148.729
C03142=1170.884,163.552,-57.169,-178.312,6.663,148.729
C03143=1170.880,163.802,-57.192,-178.309,6.664,148.728
C03144=1170.874,164.051,-57.212,-178.306,6.666,148.728
C03145=1170.870,164.300,-57.235,-178.304,6.668,148.727
C03146=1170.865,164.549,-57.256,-178.301,6.670,148.727
C03147=1170.860,164.798,-57.278,-178.298,6.671,148.727
C03148=1170.855,165.047,-57.301,-178.296,6.673,148.726
C03149=1170.851,165.296,-57.322,-178.293,6.675,148.726
C03150=1170.846,165.545,-57.344,-178.290,6.677,148.726
C03151=1170.841,165.794,-57.366,-178.288,6.678,148.725
C03152=1170.837,166.043,-57.388,-178.285,6.680,148.725
C03153=1170.832,166.292,-57.410,-178.282,6.683,148.725
C03154=1170.828,166.541,-57.432,-178.279,6.685,148.724
C03155=1170.823,166.790,-57.453,-178.277,6.687,148.724
C03156=1170.819,167.039,-57.477,-178.274,6.688,148.724
C03157=1170.814,167.287,-57.498,-178.271,6.690,148.723
C03158=1170.809,167.537,-57.521,-178.269,6.692,148.723
C03159=1170.804,167.785,-57.542,-178.266,6.694,148.723
C03160=1170.800,168.035,-57.564,-178.263,6.695,148.722
C03161=1170.795,168.284,-57.587,-178.261,6.697,148.722
C03162=1170.790,168.533,-57.609,-178.258,6.699,148.721
C03163=1170.785,168.782,-57.630,-178.255,6.701,148.721
C03164=1170.781,169.031,-57.652,-178.252,6.704,148.721
C03165=1170.777,169.279,-57.675,-178.250,6.705,148.721
C03166=1170.772,169.529,-57.697,-178.247,6.707,148.720
C03167=1170.767,169.777,-57.719,-178.244,6.709,148.720
C03168=1170.763,170.027,-57.741,-178.242,6.711,148.719
C03169=1170.758,170.275,-57.763,-178.239,6.712,148.719
C03170=1170.753,170.524,-57.786,-178.236,6.714,148.719
C03171=1170.748,170.773,-57.808,-178.234,6.716,148.718
C03172=1170.744,171.022,-57.830,-178.230,6.718,148.718
C03173=1170.739,171.272,-57.852,-178.228,6.720,148.718
C03174=1170.734,171.520,-57.875,-178.225,6.722,148.718
C03175=1170.730,171.769,-57.897,-178.223,6.724,148.717
C03176=1170.725,172.018,-57.919,-178.220,6.726,148.717
C03177=1170.720,172.267,-57.942,-178.217,6.728,148.716
C03178=1170.716,172.516,-57.964,-178.215,6.729,148.716
C03179=1170.711,172.765,-57.986,-178.211,6.732,148.716
C03180=1170.707,173.014,-58.009,-178.209,6.734,148.715
C03181=1170.702,173.263,-58.031,-178.206,6.735,148.715
C03182=1170.697,173.512,-58.053,-178.204,6.738,148.715
C03183=1170.693,173.761,-58.076,-178.201,6.739,148.714
C03184=1170.688,174.010,-58.098,-178.199,6.741,148.714
C03185=1170.683,174.259,-58.120,-178.196,6.743,148.714
C03186=1170.678,174.507,-58.143,-178.193,6.745,148.713
C03187=1170.674,174.757,-58.165,-178.190,6.747,148.713
C03188=1170.669,175.006,-58.188,-178.187,6.749,148.713
C03189=1170.664,175.254,-58.210,-178.185,6.751,148.712
C03190=1170.660,175.503,-58.233,-178.182,6.753,148.712
C03191=1170.655,175.753,-58.255,-178.180,6.755,148.712
C03192=1170.651,176.001,-58.278,-178.177,6.756,148.711
C03193=1170.646,176.250,-58.300,-178.174,6.759,148.711
C03194=1170.642,176.499,-58.323,-178.171,6.761,148.711
C03195=1170.636,176.748,-58.345,-178.168,6.762,148.710
C03196=1170.632,176.997,-58.368,-178.166,6.764,148.710
C03197=1170.627,177.247,-58.391,-178.163,6.766,148.710
C03198=1170.623,177.495,-58.413,-178.161,6.768,148.709
C03199=1170.618,177.744,-58.436,-178.158,6.771,148.709
C03200=1170.614,177.993,-58.459,-178.155,6.772,148.709
C03201=1170.608,178.242,-58.481,-178.152,6.774,148.708
C03202=1170.604,178.491,-58.504,-178.149,6.776,148.708
C03203=1170.600,178.740,-58.527,-178.147,6.778,148.708
C03204=1170.595,178.989,-58.549,-178.144,6.781,148.708
C03205=1170.590,179.237,-58.572,-178.141,6.782,148.707
C03206=1170.586,179.487,-58.594,-178.139,6.784,148.707
C03207=1170.581,179.736,-58.618,-178.136,6.786,148.707
C03208=1170.577,179.984,-58.640,-178.133,6.788,148.706
C03209=1170.571,180.233,-58.663,-178.131,6.790,148.706
C03210=1170.568,180.482,-58.685,-178.128,6.792,148.706
C03211=1170.563,180.731,-58.709,-178.125,6.794,148.705
C03212=1170.558,180.980,-58.732,-178.122,6.796,148.705
C03213=1170.553,181.229,-58.754,-178.120,6.798,148.705
C03214=1170.549,181.478,-58.777,-178.118,6.800,148.704
C03215=1170.545,181.727,-58.800,-178.114,6.802,148.704
C03216=1170.540,181.976,-58.822,-178.112,6.804,148.704
C03217=1170.534,182.224,-58.845,-178.109,6.806,148.703
C03218=1170.530,182.473,-58.868,-178.106,6.808,148.703
C03219=1170.526,182.722,-58.892,-178.104,6.810,148.703
C03220=1170.521,182.971,-58.915,-178.101,6.812,148.703
C03221=1170.517,183.221,-58.937,-178.098,6.814,148.702
C03222=1170.511,183.469,-58.960,-178.095,6.816,148.702
C03223=1170.507,183.718,-58.983,-178.093,6.818,148.701
C03224=1170.502,183.987,-59.008,-178.090,6.820,148.701
C03225=1170.497,184.257,-59.033,-178.087,6.822,148.701
C03226=1170.492,184.527,-59.057,-178.084,6.825,148.701
C03227=1170.487,184.796,-59.083,-178.081,6.827,148.700
C03228=1170.482,185.045,-59.106,-178.078,6.829,148.700
C03229=1170.477,185.294,-59.129,-178.075,6.831,148.700
C03230=1170.473,185.543,-59.152,-178.073,6.833,148.699
C03231=1170.469,185.792,-59.175,-178.070,6.835,148.699
C03232=1170.464,186.041,-59.199,-178.068,6.837,148.699
C03233=1170.460,186.290,-59.221,-178.065,6.839,148.698
C03234=1170.455,186.538,-59.244,-178.062,6.841,148.698
C03235=1170.450,186.787,-59.268,-178.059,6.843,148.698
C03236=1170.445,187.036,-59.291,-178.057,6.845,148.698
C03237=1170.441,187.285,-59.314,-178.054,6.848,148.697
C03238=1170.437,187.534,-59.337,-178.051,6.849,148.697
C03239=1170.432,187.783,-59.360,-178.049,6.851,148.697
C03240=1170.427,188.032,-59.384,-178.046,6.853,148.696
C03241=1170.423,188.281,-59.407,-178.043,6.856,148.696
C03242=1170.418,188.530,-59.431,-178.040,6.858,148.696
C03243=1170.413,188.778,-59.453,-178.038,6.859,148.695
C03244=1170.409,189.027,-59.476,-178.035,6.861,148.695
C03245=1170.404,189.276,-59.500,-178.032,6.864,148.695
C03246=1170.400,189.525,-59.524,-178.030,6.866,148.695
C03247=1170.395,189.774,-59.547,-178.027,6.868,148.694
C03248=1170.390,190.023,-59.570,-178.024,6.870,148.694
C03249=1170.385,190.272,-59.594,-178.021,6.872,148.694
C03250=1170.381,190.521,-59.617,-178.019,6.874,148.693
C03251=1170.377,190.770,-59.640,-178.016,6.876,148.693
C03252=1170.372,191.018,-59.664,-178.014,6.878,148.693
C03253=1170.368,191.267,-59.687,-178.011,6.881,148.693
C03254=1170.363,191.516,-59.711,-178.008,6.882,148.692
C03255=1170.358,191.765,-59.734,-178.005,6.884,148.692
C03256=1170.354,192.014,-59.757,-178.003,6.887,148.692
C03257=1170.349,192.263,-59.782,-178.000,6.889,148.691
C03258=1170.345,192.512,-59.805,-177.997,6.891,148.691
C03259=1170.340,192.761,-59.828,-177.994,6.893,148.691
C03260=1170.335,193.010,-59.852,-177.992,6.895,148.691
C03261=1170.331,193.258,-59.876,-177.989,6.897,148.690
C03262=1170.326,193.507,-59.899,-177.986,6.899,148.690
C03263=1170.321,193.756,-59.922,-177.984,6.902,148.690
C03264=1170.317,194.005,-59.946,-177.981,6.904,148.689
C03265=1170.312,194.254,-59.970,-177.978,6.905,148.689
C03266=1170.308,194.503,-59.993,-177.976,6.907,148.689
C03267=1170.303,194.751,-60.017,-177.973,6.910,148.689
C03268=1170.298,195.000,-60.041,-177.970,6.912,148.688
C03269=1170.294,195.249,-60.064,-177.967,6.914,148.688
C03270=1170.289,195.498,-60.088,-177.965,6.917,148.688
C03271=1170.285,195.747,-60.111,-177.962,6.918,148.687
C03272=1170.280,195.995,-60.135,-177.959,6.920,148.687
C03273=1170.276,196.244,-60.159,-177.956,6.923,148.687
C03274=1170.271,196.493,-60.182,-177.954,6.925,148.687
C03275=1170.266,196.741,-60.206,-177.951,6.927,148.686
C03276=1170.262,196.990,-60.230,-177.949,6.929,148.686
C03277=1170.257,197.239,-60.254,-177.946,6.931,148.686
C03278=1170.252,197.488,-60.278,-177.943,6.933,148.685
C03279=1170.248,197.737,-60.302,-177.940,6.935,148.685
C03280=1170.243,197.986,-60.325,-177.938,6.938,148.685
C03281=1170.239,198.235,-60.350,-177.935,6.940,148.685
C03282=1170.234,198.484,-60.373,-177.932,6.941,148.684
C03283=1170.230,198.732,-60.397,-177.930,6.944,148.684
C03284=1170.225,198.981,-60.420,-177.927,6.946,148.684
C03285=1170.221,199.230,-60.444,-177.924,6.948,148.684
C03286=1170.216,199.478,-60.469,-177.921,6.951,148.683
C03287=1170.211,199.727,-60.492,-177.919,6.953,148.683
C03288=1170.207,199.976,-60.516,-177.916,6.954,148.683
C03289=1170.203,200.226,-60.540,-177.913,6.957,148.683
C03290=1170.198,200.474,-60.564,-177.911,6.959,148.682
C03291=1170.193,200.723,-60.589,-177.908,6.961,148.682
C03292=1170.188,200.972,-60.612,-177.905,6.964,148.682
C03293=1170.184,201.220,-60.636,-177.902,6.966,148.682
C03294=1170.180,201.469,-60.660,-177.900,6.967,148.681
C03295=1170.175,201.718,-60.684,-177.897,6.970,148.681
C03296=1170.170,201.967,-60.709,-177.894,6.972,148.681
C03297=1170.166,202.215,-60.733,-177.892,6.974,148.680
C03298=1170.161,202.464,-60.756,-177.889,6.977,148.680
C03299=1170.157,202.713,-60.780,-177.886,6.979,148.680
C03300=1170.152,202.962,-60.805,-177.884,6.980,148.680
C03301=1170.148,203.211,-60.829,-177.881,6.983,148.679
C03302=1170.144,203.459,-60.854,-177.878,6.985,148.679
C03303=1170.138,203.708,-60.878,-177.875,6.988,148.679
C03304=1170.134,203.957,-60.902,-177.873,6.990,148.679
C03305=1170.130,204.206,-60.926,-177.870,6.992,148.678
C03306=1170.125,204.455,-60.951,-177.867,6.995,148.678
C03307=1170.120,204.703,-60.975,-177.865,6.996,148.678
C03308=1170.116,204.952,-60.998,-177.862,6.998,148.678
C03309=1170.111,205.201,-61.023,-177.859,7.001,148.677
C03310=1170.107,205.450,-61.047,-177.856,7.003,148.677
C03311=1170.102,205.698,-61.071,-177.854,7.005,148.677
C03312=1170.097,205.947,-61.096,-177.851,7.008,148.677
C03313=1170.093,206.196,-61.120,-177.848,7.009,148.676
C03314=1170.088,206.445,-61.145,-177.846,7.012,148.676
C03315=1170.084,206.693,-61.169,-177.843,7.014,148.676
C03316=1170.079,206.942,-61.193,-177.840,7.016,148.676
C03317=1170.075,207.191,-61.218,-177.838,7.019,148.675
C03318=1170.070,207.440,-61.242,-177.835,7.021,148.675
C03319=1170.065,207.689,-61.266,-177.833,7.023,148.675
C03320=1170.061,207.937,-61.290,-177.829,7.025,148.675
C03321=1170.056,208.187,-61.315,-177.827,7.027,148.674
C03322=1170.052,208.435,-61.339,-177.824,7.030,148.674
C03323=1170.047,208.684,-61.364,-177.821,7.032,148.674
C03324=1170.043,208.933,-61.389,-177.819,7.034,148.674
C03325=1170.039,209.181,-61.413,-177.816,7.037,148.673
C03326=1170.034,209.430,-61.438,-177.813,7.038,148.673
C03327=1170.030,209.679,-61.463,-177.810,7.041,148.673
C03328=1170.025,209.949,-61.489,-177.808,7.043,148.673
C03329=1170.019,210.220,-61.515,-177.805,7.046,148.672
C03330=1170.015,210.491,-61.542,-177.802,7.049,148.672
C03331=1170.010,210.761,-61.569,-177.799,7.050,148.672
C03332=1170.004,211.009,-61.594,-177.796,7.053,148.672
C03333=1170.001,211.259,-61.618,-177.794,7.055,148.671
C03334=1169.996,211.507,-61.643,-177.790,7.058,148.671
C03335=1169.991,211.755,-61.668,-177.788,7.060,148.671
C03336=1169.987,212.004,-61.693,-177.785,7.063,148.671
C03337=1169.982,212.253,-61.717,-177.783,7.065,148.671
C03338=1169.978,212.502,-61.742,-177.780,7.066,148.670
C03339=1169.973,212.750,-61.767,-177.777,7.069,148.670
C03340=1169.969,212.999,-61.791,-177.775,7.071,148.670
C03341=1169.964,213.248,-61.816,-177.771,7.074,148.670
C03342=1169.959,213.497,-61.841,-177.769,7.076,148.669
C03343=1169.956,213.745,-61.866,-177.766,7.079,148.669
C03344=1169.950,213.994,-61.891,-177.764,7.081,148.669
C03345=1169.946,214.243,-61.915,-177.761,7.082,148.669
C03346=1169.942,214.492,-61.940,-177.758,7.085,148.669
C03347=1169.937,214.740,-61.965,-177.756,7.087,148.668
C03348=1169.933,214.989,-61.990,-177.752,7.090,148.668
C03349=1169.928,215.238,-62.014,-177.750,7.092,148.668
C03350=1169.924,215.487,-62.040,-177.747,7.095,148.667
C03351=1169.919,215.735,-62.064,-177.745,7.097,148.667
C03352=1169.914,215.983,-62.090,-177.742,7.098,148.667
C03353=1169.910,216.233,-62.115,-177.739,7.101,148.667
C03354=1169.905,216.481,-62.139,-177.737,7.103,148.667
C03355=1169.901,216.730,-62.164,-177.734,7.106,148.667
C03356=1169.896,216.979,-62.189,-177.731,7.108,148.666
C03357=1169.892,217.227,-62.215,-177.729,7.111,148.666
C03358=1169.887,217.476,-62.239,-177.726,7.113,148.666
C03359=1169.883,217.725,-62.265,-177.723,7.116,148.666
C03360=1169.878,217.973,-62.289,-177.720,7.117,148.665
C03361=1169.874,218.222,-62.315,-177.718,7.120,148.665
C03362=1169.869,218.471,-62.340,-177.715,7.122,148.665
C03363=1169.865,218.719,-62.365,-177.712,7.125,148.665
C03364=1169.860,218.968,-62.390,-177.710,7.127,148.664
C03365=1169.856,219.217,-62.415,-177.707,7.129,148.664
C03366=1169.851,219.466,-62.440,-177.704,7.132,148.664
C03367=1169.847,219.714,-62.466,-177.702,7.134,148.664
C03368=1169.843,219.964,-62.490,-177.699,7.136,148.664
C03369=1169.838,220.212,-62.516,-177.697,7.138,148.664
C03370=1169.834,220.461,-62.541,-177.693,7.141,148.663
C03371=1169.829,220.709,-62.566,-177.691,7.143,148.663
C03372=1169.824,220.958,-62.592,-177.688,7.146,148.663
C03373=1169.819,221.207,-62.616,-177.686,7.148,148.663
C03374=1169.816,221.455,-62.642,-177.682,7.151,148.662
C03375=1169.811,221.703,-62.667,-177.680,7.153,148.662
C03376=1169.806,221.953,-62.692,-177.677,7.155,148.662
C03377=1169.802,222.202,-62.718,-177.675,7.157,148.662
C03378=1169.797,222.450,-62.743,-177.672,7.160,148.662
C03379=1169.793,222.699,-62.768,-177.669,7.162,148.661
C03380=1169.788,222.947,-62.794,-177.666,7.165,148.661
C03381=1169.784,223.196,-62.819,-177.664,7.167,148.661
C03382=1169.779,223.445,-62.845,-177.661,7.169,148.661
C03383=1169.774,223.694,-62.870,-177.659,7.172,148.661
C03384=1169.770,223.942,-62.895,-177.655,7.174,148.660
C03385=1169.765,224.190,-62.921,-177.653,7.176,148.660
C03386=1169.761,224.439,-62.947,-177.650,7.179,148.660
C03387=1169.757,224.688,-62.972,-177.648,7.181,148.660
C03388=1169.752,224.937,-62.997,-177.645,7.184,148.660
C03389=1169.748,225.186,-63.023,-177.642,7.186,148.659
C03390=1169.743,225.434,-63.048,-177.640,7.189,148.659
C03391=1169.738,225.683,-63.074,-177.637,7.191,148.659
C03392=1169.734,225.931,-63.100,-177.634,7.194,148.659
C03393=1169.730,226.180,-63.125,-177.631,7.195,148.659
C03394=1169.725,226.428,-63.151,-177.629,7.198,148.658
C03395=1169.721,226.678,-63.176,-177.625,7.201,148.658
C03396=1169.716,226.926,-63.202,-177.623,7.203,148.658
C03397=1169.712,227.175,-63.227,-177.621,7.206,148.658
C03398=1169.707,227.423,-63.253,-177.618,7.208,148.658
C03399=1169.703,227.672,-63.278,-177.615,7.211,148.658
C03400=1169.698,227.920,-63.304,-177.612,7.212,148.657
C03401=1169.694,228.169,-63.330,-177.610,7.215,148.657
C03402=1169.690,228.418,-63.355,-177.607,7.217,148.657
C03403=1169.685,228.666,-63.381,-177.604,7.220,148.657
C03404=1169.680,228.915,-63.407,-177.602,7.222,148.657
C03405=1169.676,229.164,-63.433,-177.599,7.225,148.656
C03406=1169.672,229.413,-63.459,-177.597,7.227,148.656
C03407=1169.667,229.661,-63.484,-177.593,7.230,148.656
C03408=1169.663,229.910,-63.510,-177.591,7.233,148.656
C03409=1169.658,230.158,-63.535,-177.588,7.235,148.656
C03410=1169.654,230.407,-63.562,-177.585,7.237,148.655
C03411=1169.649,230.655,-63.588,-177.583,7.240,148.655
C03412=1169.645,230.904,-63.614,-177.580,7.242,148.655
C03413=1169.640,231.153,-63.639,-177.578,7.244,148.655
C03414=1169.636,231.401,-63.665,-177.575,7.247,148.655
C03415=1169.631,231.650,-63.691,-177.572,7.249,148.654
C03416=1169.626,231.899,-63.717,-177.569,7.252,148.654
C03417=1169.622,232.147,-63.743,-177.566,7.255,148.654
C03418=1169.618,232.396,-63.769,-177.564,7.257,148.654
C03419=1169.614,232.644,-63.795,-177.561,7.260,148.654
C03420=1169.608,232.893,-63.821,-177.559,7.261,148.654
C03421=1169.604,233.142,-63.847,-177.556,7.264,148.654
C03422=1169.600,233.390,-63.873,-177.553,7.267,148.653
C03423=1169.596,233.639,-63.899,-177.550,7.269,148.653
C03424=1169.591,233.888,-63.925,-177.548,7.272,148.653
C03425=1169.586,234.136,-63.951,-177.545,7.274,148.653
C03426=1169.582,234.384,-63.977,-177.542,7.277,148.653
C03427=1169.577,234.633,-64.003,-177.540,7.279,148.653
C03428=1169.573,234.882,-64.029,-177.537,7.282,148.652
C03429=1169.569,235.130,-64.056,-177.534,7.285,148.652
C03430=1169.564,235.379,-64.082,-177.532,7.287,148.652
C03431=1169.560,235.627,-64.107,-177.529,7.289,148.652
C03432=1169.555,235.899,-64.136,-177.526,7.292,148.652
C03433=1169.550,236.171,-64.165,-177.523,7.295,148.651
C03434=1169.545,236.442,-64.193,-177.520,7.298,148.651
C03435=1169.540,236.714,-64.223,-177.517,7.300,148.651
C03436=1169.536,236.963,-64.249,-177.515,7.303,148.651
C03437=1169.532,237.211,-64.274,-177.512,7.306,148.651
C03438=1169.527,237.460,-64.301,-177.510,7.308,148.651
C03439=1169.523,237.709,-64.327,-177.506,7.310,148.650
C03440=1169.518,237.957,-64.354,-177.504,7.313,148.650
C03441=1169.514,238.206,-64.380,-177.501,7.315,148.650
C03442=1169.509,238.453,-64.406,-177.498,7.318,148.650
C03443=1169.504,238.703,-64.432,-177.496,7.320,148.650
C03444=1169.501,238.951,-64.459,-177.493,7.323,148.650
C03445=1169.496,239.200,-64.485,-177.490,7.326,148.650
C03446=1169.492,239.448,-64.512,-177.488,7.328,148.649
C03447=1169.487,239.697,-64.538,-177.485,7.331,148.649
C03448=1169.483,239.945,-64.564,-177.482,7.333,148.649
C03449=1169.478,240.194,-64.591,-177.480,7.336,148.649
C03450=1169.474,240.443,-64.617,-177.477,7.339,148.649
C03451=1169.469,240.691,-64.644,-177.475,7.341,148.649
C03452=1169.465,240.940,-64.670,-177.471,7.343,148.648
C03453=1169.460,241.188,-64.697,-177.469,7.346,148.648
C03454=1169.456,241.437,-64.724,-177.467,7.348,148.648
C03455=1169.452,241.686,-64.750,-177.463,7.351,148.648
C03456=1169.448,241.934,-64.776,-177.461,7.354,148.648
C03457=1169.443,242.182,-64.803,-177.458,7.356,148.648
C03458=1169.438,242.432,-64.830,-177.456,7.359,148.648
C03459=1169.434,242.680,-64.856,-177.452,7.362,148.648
C03460=1169.429,242.928,-64.883,-177.450,7.364,148.647
C03461=1169.425,243.176,-64.910,-177.447,7.367,148.647
C03462=1169.421,243.426,-64.936,-177.445,7.370,148.647
C03463=1169.416,243.674,-64.963,-177.442,7.372,148.647
C03464=1169.412,243.922,-64.990,-177.439,7.374,148.647
C03465=1169.407,244.171,-65.017,-177.437,7.377,148.647
C03466=1169.403,244.419,-65.043,-177.434,7.379,148.646
C03467=1169.398,244.668,-65.070,-177.431,7.382,148.646
C03468=1169.394,244.916,-65.097,-177.429,7.384,148.646
C03469=1169.390,245.165,-65.123,-177.426,7.387,148.646
C03470=1169.385,245.413,-65.150,-177.423,7.390,148.646
C03471=1169.381,245.662,-65.177,-177.421,7.392,148.646
C03472=1169.377,245.910,-65.204,-177.418,7.395,148.646
C03473=1169.372,246.158,-65.231,-177.415,7.398,148.646
C03474=1169.367,246.407,-65.257,-177.412,7.401,148.646
C03475=1169.362,246.656,-65.284,-177.410,7.403,148.645
C03476=1169.359,246.905,-65.311,-177.407,7.406,148.645
C03477=1169.354,247.153,-65.338,-177.404,7.409,148.645
C03478=1169.350,247.402,-65.365,-177.402,7.411,148.645
C03479=1169.346,247.650,-65.392,-177.399,7.413,148.645
C03480=1169.341,247.899,-65.419,-177.396,7.416,148.645
C03481=1169.336,248.147,-65.446,-177.394,7.418,148.645
C03482=1169.332,248.396,-65.473,-177.391,7.421,148.645
C03483=1169.327,248.644,-65.500,-177.388,7.424,148.645
C03484=1169.323,248.892,-65.526,-177.386,7.426,148.644
C03485=1169.319,249.141,-65.554,-177.383,7.429,148.644
C03486=1169.315,249.390,-65.581,-177.380,7.432,148.644
C03487=1169.310,249.638,-65.608,-177.378,7.434,148.644
C03488=1169.305,249.887,-65.635,-177.375,7.437,148.644
C03489=1169.301,250.135,-65.661,-177.372,7.440,148.644
C03490=1169.297,250.383,-65.689,-177.369,7.443,148.644
C03491=1169.292,250.631,-65.716,-177.367,7.445,148.643
C03492=1169.288,250.881,-65.744,-177.364,7.448,148.643
C03493=1169.284,251.129,-65.771,-177.362,7.451,148.643
C03494=1169.279,251.378,-65.798,-177.360,7.453,148.643
C03495=1169.274,251.626,-65.825,-177.356,7.456,148.643
C03496=1169.271,251.874,-65.852,-177.354,7.459,148.643
C03497=1169.267,252.123,-65.879,-177.351,7.461,148.643
C03498=1169.262,252.371,-65.906,-177.349,7.464,148.643
C03499=1169.257,252.620,-65.934,-177.346,7.467,148.643
C03500=1169.253,252.868,-65.961,-177.343,7.470,148.643
C03501=1169.248,253.116,-65.988,-177.340,7.471,148.642
C03502=1169.244,253.365,-66.016,-177.338,7.474,148.642
C03503=1169.240,253.614,-66.043,-177.335,7.477,148.642
C03504=1169.235,253.862,-66.070,-177.332,7.480,148.642
C03505=1169.231,254.110,-66.098,-177.330,7.482,148.642
C03506=1169.226,254.360,-66.125,-177.327,7.485,148.642
C03507=1169.222,254.608,-66.152,-177.324,7.488,148.642
C03508=1169.217,254.856,-66.180,-177.322,7.490,148.642
C03509=1169.213,255.104,-66.207,-177.319,7.493,148.642
C03510=1169.209,255.354,-66.234,-177.316,7.496,148.641
C03511=1169.204,255.601,-66.262,-177.314,7.499,148.641
C03512=1169.200,255.850,-66.289,-177.311,7.501,148.641
C03513=1169.195,256.098,-66.317,-177.309,7.504,148.641
C03514=1169.191,256.347,-66.344,-177.306,7.507,148.641
C03515=1169.187,256.596,-66.372,-177.303,7.510,148.641
C03516=1169.182,256.843,-66.399,-177.301,7.512,148.641
C03517=1169.178,257.092,-66.426,-177.298,7.515,148.641
C03518=1169.174,257.340,-66.455,-177.295,7.518,148.641
C03519=1169.169,257.589,-66.482,-177.292,7.521,148.641
C03520=1169.165,257.837,-66.509,-177.290,7.523,148.641
C03521=1169.161,258.086,-66.537,-177.287,7.526,148.641
C03522=1169.157,258.334,-66.565,-177.285,7.529,148.640
C03523=1169.151,258.583,-66.592,-177.282,7.532,148.640
C03524=1169.147,258.831,-66.620,-177.280,7.534,148.640
C03525=1169.143,259.080,-66.647,-177.277,7.537,148.640
C03526=1169.138,259.328,-66.675,-177.274,7.540,148.640
C03527=1169.135,259.576,-66.703,-177.271,7.542,148.640
C03528=1169.130,259.825,-66.730,-177.269,7.545,148.640
C03529=1169.126,260.073,-66.758,-177.266,7.548,148.640
C03530=1169.121,260.322,-66.786,-177.263,7.551,148.640
C03531=1169.116,260.570,-66.814,-177.260,7.554,148.640
C03532=1169.113,260.819,-66.842,-177.258,7.556,148.640
C03533=1169.108,261.067,-66.869,-177.256,7.559,148.640
C03534=1169.104,261.315,-66.897,-177.253,7.562,148.639
C03535=1169.099,261.564,-66.926,-177.250,7.565,148.639
C03536=1169.094,261.836,-66.956,-177.247,7.567,148.639
C03537=1169.090,262.109,-66.986,-177.245,7.570,148.639
C03538=1169.085,262.383,-67.017,-177.241,7.573,148.639
C03539=1169.080,262.656,-67.048,-177.239,7.576,148.639
C03540=1169.076,262.904,-67.076,-177.236,7.579,148.639
C03541=1169.072,263.153,-67.104,-177.233,7.582,148.639
C03542=1169.067,263.401,-67.131,-177.230,7.585,148.639
C03543=1169.062,263.650,-67.159,-177.228,7.588,148.639
C03544=1169.058,263.898,-67.188,-177.225,7.590,148.639
C03545=1169.054,264.146,-67.215,-177.223,7.593,148.639
C03546=1169.050,264.395,-67.244,-177.220,7.596,148.639
C03547=1169.045,264.643,-67.271,-177.217,7.599,148.639
C03548=1169.041,264.892,-67.299,-177.214,7.602,148.638
C03549=1169.036,265.140,-67.328,-177.212,7.604,148.638
C03550=1169.032,265.389,-67.356,-177.209,7.607,148.638
C03551=1169.028,265.637,-67.384,-177.207,7.610,148.638
C03552=1169.023,265.885,-67.412,-177.204,7.613,148.638
C03553=1169.019,266.133,-67.440,-177.201,7.616,148.638
C03554=1169.015,266.381,-67.468,-177.199,7.618,148.638
C03555=1169.010,266.630,-67.497,-177.196,7.621,148.638
C03556=1169.006,266.878,-67.524,-177.194,7.624,148.638
C03557=1169.001,267.127,-67.553,-177.191,7.627,148.638
C03558=1168.997,267.375,-67.581,-177.188,7.630,148.638
C03559=1168.993,267.623,-67.609,-177.186,7.632,148.638
C03560=1168.988,267.872,-67.637,-177.183,7.635,148.638
C03561=1168.984,268.120,-67.666,-177.180,7.638,148.638
C03562=1168.980,268.369,-67.694,-177.178,7.641,148.638
C03563=1168.976,268.617,-67.722,-177.175,7.644,148.638
C03564=1168.971,268.866,-67.751,-177.173,7.646,148.637
C03565=1168.967,269.114,-67.779,-177.170,7.649,148.637
C03566=1168.962,269.363,-67.807,-177.167,7.652,148.637
C03567=1168.958,269.610,-67.835,-177.164,7.655,148.637
C03568=1168.953,269.859,-67.864,-177.162,7.658,148.637
C03569=1168.949,270.107,-67.892,-177.159,7.661,148.637
C03570=1168.945,270.356,-67.920,-177.157,7.663,148.637
C03571=1168.941,270.604,-67.949,-177.154,7.666,148.637
C03572=1168.936,270.852,-67.978,-177.151,7.669,148.637
C03573=1168.932,271.101,-68.006,-177.148,7.672,148.637
C03574=1168.927,271.349,-68.034,-177.146,7.675,148.637
C03575=1168.924,271.598,-68.062,-177.143,7.678,148.637
C03576=1168.919,271.846,-68.092,-177.141,7.680,148.637
C03577=1168.915,272.094,-68.119,-177.138,7.683,148.637
C03578=1168.910,272.343,-68.148,-177.135,7.686,148.637
C03579=1168.905,272.591,-68.177,-177.133,7.689,148.637
C03580=1168.902,272.839,-68.205,-177.130,7.692,148.637
C03581=1168.897,273.088,-68.234,-177.128,7.695,148.637
C03582=1168.893,273.335,-68.262,-177.125,7.698,148.637
C03583=1168.889,273.584,-68.291,-177.123,7.700,148.637
C03584=1168.884,273.833,-68.320,-177.120,7.703,148.637
C03585=1168.880,274.081,-68.348,-177.117,7.706,148.637
C03586=1168.876,274.329,-68.377,-177.114,7.709,148.637
C03587=1168.871,274.578,-68.406,-177.112,7.712,148.636
C03588=1168.867,274.826,-68.434,-177.109,7.715,148.636
C03589=1168.863,275.074,-68.463,-177.106,7.718,148.636
C03590=1168.858,275.323,-68.492,-177.104,7.720,148.636
C03591=1168.854,275.570,-68.521,-177.101,7.723,148.636
C03592=1168.850,275.819,-68.549,-177.098,7.726,148.636
C03593=1168.845,276.068,-68.578,-177.096,7.729,148.636
C03594=1168.841,276.315,-68.607,-177.093,7.732,148.636
C03595=1168.837,276.564,-68.635,-177.091,7.735,148.636
C03596=1168.833,276.812,-68.665,-177.088,7.738,148.636
C03597=1168.828,277.060,-68.693,-177.086,7.740,148.636
C03598=1168.824,277.308,-68.722,-177.083,7.743,148.636
C03599=1168.820,277.557,-68.751,-177.080,7.746,148.636
C03600=1168.815,277.805,-68.780,-177.077,7.749,148.636
C03601=1168.811,278.053,-68.809,-177.075,7.752,148.636
C03602=1168.807,278.302,-68.837,-177.072,7.756,148.636
C03603=1168.803,278.550,-68.867,-177.070,7.759,148.636
C03604=1168.798,278.799,-68.896,-177.067,7.762,148.636
C03605=1168.793,279.046,-68.925,-177.065,7.764,148.636
C03606=1168.789,279.295,-68.954,-177.062,7.767,148.636
C03607=1168.786,279.543,-68.982,-177.059,7.770,148.636
C03608=1168.781,279.791,-69.012,-177.057,7.773,148.636
C03609=1168.776,280.040,-69.040,-177.054,7.776,148.636
C03610=1168.772,280.288,-69.070,-177.052,7.779,148.636
C03611=1168.768,280.536,-69.099,-177.049,7.782,148.636
C03612=1168.764,280.784,-69.128,-177.046,7.785,148.636
C03613=1168.759,281.033,-69.157,-177.043,7.788,148.636
C03614=1168.755,281.281,-69.186,-177.041,7.790,148.636
C03615=1168.751,281.529,-69.215,-177.038,7.793,148.636
C03616=1168.747,281.778,-69.244,-177.036,7.796,148.636
C03617=1168.742,282.026,-69.273,-177.033,7.799,148.636
C03618=1168.738,282.274,-69.303,-177.031,7.802,148.636
C03619=1168.733,282.522,-69.332,-177.028,7.805,148.636
C03620=1168.729,282.770,-69.361,-177.025,7.808,148.636
C03621=1168.725,283.019,-69.390,-177.022,7.811,148.636
C03622=1168.721,283.267,-69.419,-177.020,7.814,148.636
C03623=1168.716,283.515,-69.449,-177.017,7.817,148.636
C03624=1168.712,283.764,-69.478,-177.015,7.819,148.636
C03625=1168.707,284.011,-69.507,-177.012,7.822,148.636
C03626=1168.703,284.260,-69.537,-177.010,7.825,148.636
C03627=1168.699,284.508,-69.566,-177.007,7.828,148.636
C03628=1168.695,284.757,-69.595,-177.005,7.832,148.636
C03629=1168.690,285.005,-69.625,-177.002,7.835,148.636
C03630=1168.686,285.253,-69.654,-176.999,7.838,148.636
C03631=1168.682,285.502,-69.683,-176.996,7.841,148.636
C03632=1168.678,285.750,-69.713,-176.994,7.844,148.636
C03633=1168.674,285.998,-69.742,-176.991,7.846,148.636
C03634=1168.669,286.246,-69.771,-176.989,7.850,148.636
C03635=1168.665,286.494,-69.801,-176.986,7.853,148.636
C03636=1168.661,286.742,-69.830,-176.983,7.856,148.636
C03637=1168.656,286.990,-69.860,-176.981,7.858,148.636
C03638=1168.652,287.239,-69.889,-176.979,7.861,148.636
C03639=1168.648,287.487,-69.919,-176.976,7.864,148.636
C03640=1168.643,287.762,-69.952,-176.973,7.868,148.636
C03641=1168.638,288.037,-69.985,-176.970,7.871,148.636
C03642=1168.633,288.311,-70.018,-176.967,7.874,148.636
C03643=1168.628,288.587,-70.050,-176.964,7.878,148.636
C03644=1168.624,288.835,-70.080,-176.961,7.881,148.636
C03645=1168.620,289.083,-70.109,-176.959,7.884,148.636
C03646=1168.616,289.331,-70.139,-176.956,7.887,148.636
C03647=1168.612,289.579,-70.169,-176.954,7.889,148.636
C03648=1168.608,289.827,-70.198,-176.951,7.892,148.636
C03649=1168.603,290.076,-70.228,-176.949,7.895,148.636
C03650=1168.598,290.324,-70.258,-176.946,7.898,148.636
C03651=1168.595,290.572,-70.288,-176.943,7.901,148.636
C03652=1168.590,290.820,-70.317,-176.941,7.904,148.636
C03653=1168.586,291.068,-70.347,-176.938,7.907,148.636
C03654=1168.581,291.317,-70.377,-176.936,7.910,148.636
C03655=1168.577,291.565,-70.407,-176.933,7.913,148.636
C03656=1168.573,291.813,-70.436,-176.930,7.917,148.636
C03657=1168.569,292.061,-70.466,-176.928,7.920,148.636
C03658=1168.564,292.309,-70.497,-176.925,7.923,148.636
C03659=1168.560,292.557,-70.526,-176.922,7.926,148.636
